# B&R Automation Studio project NAELD004C00R10L518F00 (part 49)

#### Act_InitLocal.st
```iecst
(** 2019-04-16 **)
ACTION Act_InitLocal:

	//Input Reference Link To Local Variable
	p_udiRstErr ACCESS ADR(udiRstErr);
	p_bEn ACCESS ADR(bEn);
	p_bDis ACCESS ADR(bDis);
	p_bRun ACCESS ADR(bRun);
	p_bStop ACCESS ADR(bStop);
	p_bStep ACCESS ADR(bStep);

	p_sProgNm ACCESS ADR(sProgNm);
	p_bNtSettingsLoadDone ACCESS ADR(bNtSettingsLoadDone);

	pa_bMagDis ACCESS ADR(a_bMagDis);
	p_bUnloadMag ACCESS ADR(bUnloadMag);
	p_bDSAllow ACCESS ADR(bDSAllow);
	p_bPullerRotCylPrep ACCESS ADR(bPullerRotCylPrep);
	p_bPullerNoRotCylExitStartLif ACCESS ADR(bPullerNoRotCylExitStartLif);
	p_diPullerExtMaxSlt ACCESS ADR(diPullerExtMaxSlt);
	p_diPullerExtMinSlt ACCESS ADR(diPullerExtMinSlt);
	p_bLifterSafeInitialize ACCESS ADR(bLifterSafeInitialize);

	p_bProdRcpCurrRcpTopToBtm ACCESS ADR(bProdRcpCurrRcpTopToBtm);
	p_diProdRcpCurrRcpPitch ACCESS ADR(diProdRcpCurrRcpPitch);

	p_bMagSetupDone1 ACCESS ADR(bMagSetupDone1);
	p_bMagSetupDone2 ACCESS ADR(bMagSetupDone2);
	p_bMagSetupDone3 ACCESS ADR(bMagSetupDone3);

	p_tyBufferStat1 ACCESS ADR(tyBufferStat1);
	p_tyBufferStat2 ACCESS ADR(tyBufferStat2);
	p_tyBufferStat3 ACCESS ADR(tyBufferStat3);

	p_bMagPresentSen1 ACCESS ADR(bMagPresentSen1);
	p_bMagPresentSen2 ACCESS ADR(bMagPresentSen2);
	p_bMagPresentSen3 ACCESS ADR(bMagPresentSen3);

	p_bBufferMagPresent1 ACCESS ADR(bBufferMagPresent1);
	p_bBufferMagPresent2 ACCESS ADR(bBufferMagPresent2);
	p_bBufferMagPresent3 ACCESS ADR(bBufferMagPresent3);

	p_dtBufferMagPresentTm1 ACCESS ADR(dtBufferMagPresentTm1);
	p_dtBufferMagPresentTm2 ACCESS ADR(dtBufferMagPresentTm2);
	p_dtBufferMagPresentTm3 ACCESS ADR(dtBufferMagPresentTm3);

	p_eLifterStat ACCESS ADR(eLifterStat);
	p_eLifterStatus ACCESS ADR(eLifterStatus);

	p_eBufferStat1 ACCESS ADR(eBufferStat1);
	p_eBufferStatus1 ACCESS ADR(eBufferStatus1);

	p_eBufferStat2 ACCESS ADR(eBufferStat2);
	p_eBufferStatus2 ACCESS ADR(eBufferStatus2);

	p_eBufferStat3 ACCESS ADR(eBufferStat3);
	p_eBufferStatus3 ACCESS ADR(eBufferStatus3);

	p_eDSSMEMAStat1 ACCESS ADR(eDSSMEMAStat1);
	p_eDSSMEMAStatus1 ACCESS ADR(eDSSMEMAStatus1);
	p_bDSSMEMAConvStart1 ACCESS ADR(bDSSMEMAConvStart1);

	p_eDSSMEMAStat2 ACCESS ADR(eDSSMEMAStat2);
	p_eDSSMEMAStatus2 ACCESS ADR(eDSSMEMAStatus2);
	p_bDSSMEMAConvStart2 ACCESS ADR(bDSSMEMAConvStart2);

	p_eDSSMEMAStat3 ACCESS ADR(eDSSMEMAStat3);
	p_eDSSMEMAStatus3 ACCESS ADR(eDSSMEMAStatus3);
	p_bDSSMEMAConvStart3 ACCESS ADR(bDSSMEMAConvStart3);

	p_diBufferNxtUnloadSlt1 ACCESS ADR(diBufferNxtUnloadSlt1);
	p_diBufferNxtUnloadSlt2 ACCESS ADR(diBufferNxtUnloadSlt2);
	p_diBufferNxtUnloadSlt3 ACCESS ADR(diBufferNxtUnloadSlt3);

END_ACTION
```

#### Act_Link.st
```iecst
(** 2018-12-11 **)
ACTION Act_Link:
	p_bLifterSafeInitialize := p_bLinkPullerRetRS AND p_bLinkInShutterCloRS;

END_ACTION
```

#### Init.st
```iecst
(** 2019-03-25 **)
PROGRAM _INIT

	(* Always Change If Project Change *)

	//Pass Address To Global Address For External Use
	//Action, State & Status

	//Alarm
	p_OpsLifMagLDAlmData	:= ADR(tyAlmData);
	p_OpsLifMagLDAlmData1	:= ADR(tyAlmData1);

	//Output
	p_OpsLifMagLDStepTxt	:= ADR(sStepTxt);
	p_OpsLifMagLDPaused		:= ADR(bPaused);

	p_OpsLifMagLDLifterAct		:= ADR(eLifterAct);
	p_OpsLifMagLDBufferAct1		:= ADR(eBufferAct1);
	p_OpsLifMagLDBufferAct2		:= ADR(eBufferAct2);
	p_OpsLifMagLDBufferAct3		:= ADR(eBufferAct3);
	p_OpsLifMagLDDSSMEMAAct1	:= ADR(eDSSMEMAAct1);
	p_OpsLifMagLDDSSMEMAAct2	:= ADR(eDSSMEMAAct2);
	p_OpsLifMagLDDSSMEMAAct3	:= ADR(eDSSMEMAAct3);

	p_OpsLifMagLDGoUnloadSlt1	:= ADR(diGoUnloadSlt1);
	p_OpsLifMagLDGoUnloadSlt2	:= ADR(diGoUnloadSlt2);
	p_OpsLifMagLDGoUnloadSlt3	:= ADR(diGoUnloadSlt3);
	p_OpsLifMagLDMagNxtUnload	:= ADR(eMagNxtUnload);
	p_OpsLifMagLDBffrExitBrd	:= ADR(bBffrExitBrd);
	p_OpsLifMagLDUnloadingMov	:= ADR(bUnloadingMov);
	p_OpsLifMagLDUnloading		:= ADR(bUnloading);

	(* Always Change If Project Change *)

END_PROGRAM
```

#### Act_OpsInitial.st - Do Not Change!!!
```iecst
(** 2019-01-16 **)
ACTION Act_OpsInitial:

	eOpsStep		:= LifMagLDStepNA;
	eGotoOpsStep	:= LifMagLDStepInitLif;

	eOpsStep1		:= LifMagLDStep1NA;
	eGotoOpsStep1	:= LifMagLDStep1InitLif;

	eMagNxtUnload	:= MagNxtUnloadInvalid;
	bBffrExitBrd	:= FALSE;
	bUnloadingMov	:= FALSE;
	bUnloading		:= FALSE;

END_ACTION
```

#### Act_OpsRun.st
```iecst
(** 2019-04-16 **)
ACTION Act_OpsRun:

//	IF p_bPullerRotCylPrep = TRUE THEN
//		Act_OpsSubRun;
//	ELSE
		Act_OpsSubRun1;
//	END_IF

END_ACTION
```

#### Act_OpsInfo.st
```iecst
ACTION Act_OpsInfo:

	//Reset
	udiStatus1	:= 0;

	//Magazine Not Present
	a_bMagAllwMagPresent[1]	:= p_bMagPresentSen1;
	a_bMagAllwMagPresent[2]	:= p_bMagPresentSen2;
	a_bMagAllwMagPresent[3]	:= p_bMagPresentSen3;

	FOR udi := 1 TO 3 DO
		IF pa_bMagDis[udi] = FALSE AND a_bMagAllwMagPresent[udi] = TRUE THEN
			EXIT;
		END_IF
	END_FOR

	IF udi = 4 THEN
		IF (eOpsStep > LifMagLDStepInitLif) OR (eOpsStep1 > LifMagLDStep1InitLif) THEN
			udiStatus1	:= 10000;
		END_IF
	END_IF

	//Magazine Is Empty
	a_tyMagAllwBffrStat[1]	:= p_tyBufferStat1;
	a_tyMagAllwBffrStat[2]	:= p_tyBufferStat2;
	a_tyMagAllwBffrStat[3]	:= p_tyBufferStat3;

	FOR udi := 1 TO 3 DO
		IF pa_bMagDis[udi] = FALSE AND a_bMagAllwMagPresent[udi] = TRUE AND a_tyMagAllwBffrStat[udi].bBffrMty = TRUE THEN
			udiStatus1	:= 10001 + (udi - 1);
			EXIT;
		END_IF
	END_FOR

END_ACTION
```

#### Act_OpsRst.st - Do Not Change!!!
```iecst
(** 2019-03-25 **)
ACTION Act_OpsRst:

	udiStatus1	:= 0;

	eLifterAct		:= LifterActIdle;
	eBufferAct1		:= BufferActIdle;
	eBufferAct2		:= BufferActIdle;
	eBufferAct3		:= BufferActIdle;
	eDSSMEMAAct1	:= SMEMAActIdle;
	eDSSMEMAAct2	:= SMEMAActIdle;
	eDSSMEMAAct3	:= SMEMAActIdle;

END_ACTION
```

#### Act_OpsSubRun.st
```iecst
ACTION Act_OpsSubRun:

	(*Loader's Lifter Magazine Layout*)
	(*
		Direction: -->> LEFT TO RIGHT -->>

	     +----------+
	     |          |
	     |          |
	     |          |DS3 (Lif=PosCSlt)
	     |          |[Mag 3]
	     |          |
	     |          |DS2 (Lif=PosBSlt)
	     |          |[Mag 2]
	     |          |
	     |          |DS1 (Lif=PosASlt)
	     |          |[Mag 1]
	     |  Loader  |
	     +----------+

		Note: Program Action Called For Lifter As Shown Above
		      Setup Lifter Program Parameters Accordingly
	*)

	IF eGotoOpsStep <> eOpsStep THEN

		CASE eGotoOpsStep OF

			ELSE
				eOpsStep	:= eGotoOpsStep;

		END_CASE

	END_IF

	IF eOpsStep = eGotoOpsStep THEN

		IF bPaused = FALSE THEN

			CASE eOpsStep OF

				LifMagLDStepInitLif:
					sStepTxt	:= 'Initializing Lifter';

					IF p_bLifterSafeInitialize THEN
						eLifterAct	:= LifterActFullHm;

						IF p_eLifterStatus = Done AND p_eLifterStat = LifterActFullHm THEN
							eLifterAct	:= LifterActIdle;

							eGotoOpsStep	:= LifMagLDStepMagCmp;

							bPaused	:= p_bStop OR p_bStep;
						END_IF
					ELSE
						IF p_eLifterStat <> LifterActIdle THEN
							eLifterAct	:= LifterActStop;

							IF p_eLifterStatus = Done AND p_eLifterStat = LifterActStop THEN
								eLifterAct	:= LifterActIdle;

								bPaused	:= p_bStop OR p_bStep;
							END_IF
						ELSE
							bPaused	:= p_bStop OR p_bStep;
						END_IF
					END_IF

				LifMagLDStepMagCmp:
					sStepTxt	:= 'Comparing Magazine';

					a_bMagAllwMagSetupDone[1]	:= p_bMagSetupDone1;
					a_bMagAllwMagSetupDone[2]	:= p_bMagSetupDone2;
					a_bMagAllwMagSetupDone[3]	:= p_bMagSetupDone3;

					a_tyMagAllwBffrStat[1]	:= p_tyBufferStat1;
					a_tyMagAllwBffrStat[2]	:= p_tyBufferStat2;
					a_tyMagAllwBffrStat[3]	:= p_tyBufferStat3;

					a_bMagAllwMagPresent[1]	:= p_bBufferMagPresent1;
					a_bMagAllwMagPresent[2]	:= p_bBufferMagPresent2;
					a_bMagAllwMagPresent[3]	:= p_bBufferMagPresent3;

					a_udiMagAllwMagPresentTm[1]	:= DT_TO_UDINT(p_dtBufferMagPresentTm1);
					a_udiMagAllwMagPresentTm[2]	:= DT_TO_UDINT(p_dtBufferMagPresentTm2);
					a_udiMagAllwMagPresentTm[3]	:= DT_TO_UDINT(p_dtBufferMagPresentTm3);

					//Sorting Priority
					memset(ADR(a_udiMagAllwPriority), 0, SIZEOF(a_udiMagAllwPriority));

					FOR udi := 1 TO 3 DO
						udiCount	:= 3;
						udiCmpTm	:= a_udiMagAllwMagPresentTm[udi];

						FOR udi1 := 1 TO 3 DO
							IF a_udiMagAllwMagPresentTm[udi1] > udiCmpTm THEN
								udiCount	:= udiCount - 1;
							END_IF
						END_FOR

						a_udiMagAllwPriority[udi]	:= udiCount;
					END_FOR

					FOR udi := 3 TO 1 BY -1 DO
						FOR udi1 := 3 TO 1 BY -1 DO
							IF (udi <> udi1) AND (a_udiMagAllwPriority[udi] = a_udiMagAllwPriority[udi1]) THEN
								a_udiMagAllwPriority[udi1]	:= a_udiMagAllwPriority[udi1] - 1;
							END_IF
						END_FOR
					END_FOR

					//Checking Buffer Status
					memset(ADR(a_udiMagAllwSum), 0, SIZEOF(a_udiMagAllwSum));

					FOR udi := 1 TO 3 DO
						//Priority
						a_udiMagAllwSum[udi]	:= a_udiMagAllwSum[udi] + a_udiMagAllwPriority[udi];
						//Enable
						IF pa_bMagDis[udi] = FALSE THEN
							a_udiMagAllwSum[udi]	:= a_udiMagAllwSum[udi] + 1000;
						END_IF
						//Magazine Setup Complete
						IF a_bMagAllwMagSetupDone[udi] = TRUE THEN
							a_udiMagAllwSum[udi]	:= a_udiMagAllwSum[udi] + 1000;
						END_IF
						//Magazine Present
						IF a_bMagAllwMagPresent[udi] = TRUE THEN
							a_udiMagAllwSum[udi]	:= a_udiMagAllwSum[udi] + 1000;
						END_IF
						//Magazine Full
						IF a_tyMagAllwBffrStat[udi].bBffrFull = TRUE THEN
							a_udiMagAllwSum[udi]	:= a_udiMagAllwSum[udi] + 2500;
						END_IF
						//Magazine Available
						IF a_tyMagAllwBffrStat[udi].bBffrFull = FALSE AND a_tyMagAllwBffrStat[udi].bBffrMty = FALSE THEN
							a_udiMagAllwSum[udi]	:= a_udiMagAllwSum[udi] + 3000;
						END_IF

					END_FOR

					udiMagAllwGo	:= 99;

					FOR udi := 1 TO 3 DO
						//Enable + Magazine Setup Done + Magazine Present + Magazine Available
						IF a_udiMagAllwSum[udi] >= 6000 THEN

							IF udiMagAllwGo <> 99 THEN
								//Priority
								IF a_udiMagAllwSum[udi] < a_udiMagAllwSum[udiMagAllwGo] THEN
									udiMagAllwGo	:= udi;
								END_IF
							ELSE
								udiMagAllwGo	:= udi;
							END_IF

						END_IF

					END_FOR

					IF udiMagAllwGo = 99 THEN

						FOR udi := 1 TO 3 DO
							//Enable + Magazine Setup Done + Magazine Present + Magazine Full
							IF a_udiMagAllwSum[udi] >= 5500 THEN

								IF udiMagAllwGo <> 99 THEN
									//Priority
									IF a_udiMagAllwSum[udi] < a_udiMagAllwSum[udiMagAllwGo] THEN
										udiMagAllwGo	:= udi;
									END_IF
								ELSE
									udiMagAllwGo	:= udi;
								END_IF

							END_IF

						END_FOR

					END_IF

					IF (p_bDSAllow = TRUE) AND (udiMagAllwGo <> 99) THEN

						eMagNxtUnload	:= udiMagAllwGo;
						eGotoOpsStep	:= LifMagLDStepNxtUnloadBffr;

						IF eMagNxtUnload = MagNxtUnloadMag1 THEN
							p_tyLocalBufferStat ACCESS ADR(p_tyBufferStat1);
							p_bLocalBufferMagPresent ACCESS ADR(p_bBufferMagPresent1);
							p_dtLocalBufferMagPresentTm ACCESS ADR(p_dtBufferMagPresentTm1);

							p_eLocalBufferAct ACCESS ADR(eBufferAct1);
							p_eLocalBufferStat ACCESS ADR(p_eBufferStat1);
							p_eLocalBufferStatus ACCESS ADR(p_eBufferStatus1);

							p_eLocalDSSMEMAAct ACCESS ADR(eDSSMEMAAct1);
							p_eLocalDSSMEMAStat ACCESS ADR(p_eDSSMEMAStat1);
							p_eLocalDSSMEMAStatus ACCESS ADR(p_eDSSMEMAStatus1);
							p_bLocalDSSMEMAConvStart ACCESS ADR(p_bDSSMEMAConvStart1);

						ELSIF eMagNxtUnload = MagNxtUnloadMag2 THEN
							p_tyLocalBufferStat ACCESS ADR(p_tyBufferStat2);
							p_bLocalBufferMagPresent ACCESS ADR(p_bBufferMagPresent2);
							p_dtLocalBufferMagPresentTm ACCESS ADR(p_dtBufferMagPresentTm2);

							p_eLocalBufferAct ACCESS ADR(eBufferAct2);
							p_eLocalBufferStat ACCESS ADR(p_eBufferStat2);
							p_eLocalBufferStatus ACCESS ADR(p_eBufferStatus2);

							p_eLocalDSSMEMAAct ACCESS ADR(eDSSMEMAAct2);
							p_eLocalDSSMEMAStat ACCESS ADR(p_eDSSMEMAStat2);
							p_eLocalDSSMEMAStatus ACCESS ADR(p_eDSSMEMAStatus2);
							p_bLocalDSSMEMAConvStart ACCESS ADR(p_bDSSMEMAConvStart2);

						ELSIF eMagNxtUnload = MagNxtUnloadMag3 THEN
							p_tyLocalBufferStat ACCESS ADR(p_tyBufferStat3);
							p_bLocalBufferMagPresent ACCESS ADR(p_bBufferMagPresent3);
							p_dtLocalBufferMagPresentTm ACCESS ADR(p_dtBufferMagPresentTm3);

							p_eLocalBufferAct ACCESS ADR(eBufferAct3);
							p_eLocalBufferStat ACCESS ADR(p_eBufferStat3);
							p_eLocalBufferStatus ACCESS ADR(p_eBufferStatus3);

							p_eLocalDSSMEMAAct ACCESS ADR(eDSSMEMAAct3);
							p_eLocalDSSMEMAStat ACCESS ADR(p_eDSSMEMAStat3);
							p_eLocalDSSMEMAStatus ACCESS ADR(p_eDSSMEMAStatus3);
							p_bLocalDSSMEMAConvStart ACCESS ADR(p_bDSSMEMAConvStart3);

						END_IF

						bPaused	:= p_bStop OR p_bStep;

					ELSE

						eMagNxtUnload	:= MagNxtUnloadInvalid;

						bPaused	:= p_bStop;

					END_IF

					//Unload Magazine
					IF p_bUnloadMag = TRUE THEN
						eMagNxtUnload	:= MagNxtUnloadInvalid;
						eGotoOpsStep	:= LifMagLDStepLifMovUnloadMag;
					END_IF

				LifMagLDStepNxtUnloadBffr:
					sStepTxt	:= 'Computing Next Unload Buffer';

					p_eLocalBufferAct	:= BufferActNxtUnload;

					IF p_eLocalBufferStatus = Done AND p_eLocalBufferStat = BufferActNxtUnload THEN
						p_eLocalBufferAct	:= BufferActIdle;
						eGotoOpsStep		:= LifMagLDStepLifMov;

						bPaused	:= p_bStop OR p_bStep;

						//Unload Magazine
						IF p_bUnloadMag = TRUE THEN
							eMagNxtUnload	:= MagNxtUnloadInvalid;
							eGotoOpsStep	:= LifMagLDStepLifMovUnloadMag;
						END_IF

					END_IF

				LifMagLDStepLifMov:
					sStepTxt	:= 'Moving Lifter To Next Unload Position';

					diGoUnloadSlt1	:= p_diBufferNxtUnloadSlt1;
					diGoUnloadSlt2	:= p_diBufferNxtUnloadSlt2;
					diGoUnloadSlt3	:= p_diBufferNxtUnloadSlt3;

					IF eMagNxtUnload = MagNxtUnloadMag1 THEN
						eLifterAct	:= LifterActGoASltPos;

					ELSIF eMagNxtUnload = MagNxtUnloadMag2 THEN
						eLifterAct	:= LifterActGoBSltPos;

					ELSIF eMagNxtUnload = MagNxtUnloadMag3 THEN
						eLifterAct	:= LifterActGoCSltPos;

					ELSIF eMagNxtUnload = MagNxtUnloadInvalid THEN
						eGotoOpsStep	:= LifMagLDStepMagCmp;

						bPaused	:= p_bStop OR p_bStep;

						//Unload Magazine
						IF p_bUnloadMag = TRUE THEN
							eMagNxtUnload	:= MagNxtUnloadInvalid;
							eGotoOpsStep	:= LifMagLDStepLifMovUnloadMag;
						END_IF

					END_IF

					IF (p_eLifterStatus = Done AND p_eLifterStat = LifterActGoASltPos)
						OR (p_eLifterStatus = Done AND p_eLifterStat = LifterActGoBSltPos)
						OR (p_eLifterStatus = Done AND p_eLifterStat = LifterActGoCSltPos) THEN

						eLifterAct	:= LifterActIdle;

						eGotoOpsStep	:= LifMagLDStepBffrDSComm;

						bPaused	:= p_bStop OR p_bStep;

						//Unload Magazine
						IF p_bUnloadMag = TRUE THEN
							eMagNxtUnload	:= MagNxtUnloadInvalid;
							eGotoOpsStep	:= LifMagLDStepLifMovUnloadMag;
						END_IF

					END_IF

				LifMagLDStepBffrDSComm:
					sStepTxt	:= 'Communicating Buffer Downstream';

					p_eLocalDSSMEMAAct	:= SMEMAActRun;

					IF p_bLocalDSSMEMAConvStart = TRUE THEN
						eGotoOpsStep	:= LifMagLDStepBffrExitBrd;

					ELSIF p_bDSAllow = FALSE THEN
						p_eLocalDSSMEMAAct	:= SMEMAActIdle;
						eMagNxtUnload		:= MagNxtUnloadInvalid;
						eGotoOpsStep		:= LifMagLDStepMagCmp;

						bPaused	:= p_bStop OR p_bStep;

					ELSE

						IF p_bLocalBufferMagPresent = FALSE THEN	//Checking Magazine Present
							eMagNxtUnload	:= MagNxtUnloadInvalid;
							eGotoOpsStep	:= LifMagLDStepMagCmp;

							bPaused	:= p_bStop OR p_bStep;
						ELSIF pa_bMagDis[udiMagAllwGo] = TRUE THEN	//Checking Magazine Enable
							eMagNxtUnload	:= MagNxtUnloadInvalid;
							eGotoOpsStep	:= LifMagLDStepMagCmp;

							bPaused	:= p_bStop OR p_bStep;
						ELSE
							bPaused	:= p_bStop;
						END_IF

						//Unload Magazine
						IF p_bUnloadMag = TRUE THEN
							eMagNxtUnload	:= MagNxtUnloadInvalid;
							eGotoOpsStep	:= LifMagLDStepLifMovUnloadMag;

							bPaused	:= p_bStop OR p_bStep;
						END_IF

						IF (bPaused = TRUE) OR (eGotoOpsStep = LifMagLDStepMagCmp) OR (p_bUnloadMag = TRUE) THEN
							p_eLocalDSSMEMAAct	:= SMEMAActIdle;
						END_IF

					END_IF

				LifMagLDStepBffrExitBrd:
					IF p_bLocalDSSMEMAConvStart THEN
						sStepTxt	:= 'Transferring Board Out From Magazine';

						//Do Nothing
					END_IF

					IF p_eLocalDSSMEMAStatus = Done AND p_eLocalDSSMEMAStat = SMEMAActRun THEN
						p_eLocalDSSMEMAAct	:= SMEMAActIdle;
						eGotoOpsStep		:= LifMagLDStepUnloadBffr;
					END_IF

				LifMagLDStepUnloadBffr:
					sStepTxt	:= 'Unloading Buffer';

					p_eLocalBufferAct	:= BufferActUnload;

					IF p_eLocalBufferStatus = Done AND p_eLocalBufferStat = BufferActUnload THEN
						p_eLocalBufferAct	:= BufferActIdle;
						eMagNxtUnload		:= MagNxtUnloadInvalid;
						eGotoOpsStep		:= LifMagLDStepMagCmp;

						bPaused	:= p_bStop OR p_bStep;
					END_IF

				LifMagLDStepLifMovUnloadMag:
					sStepTxt	:= 'Moving Lifter To Unload Position';

					eLifterAct	:= LifterActGoAPos;

					IF p_eLifterStatus = Done AND p_eLifterStat = LifterActGoAPos THEN
						eLifterAct	:= LifterActIdle;

						eGotoOpsStep	:= LifMagLDStepUnloadMag;

						bPaused	:= p_bStop OR p_bStep;
					END_IF

				LifMagLDStepUnloadMag:
					sStepTxt	:= 'Unloading Magazine';

					IF p_bUnloadMag = FALSE THEN
						eGotoOpsStep	:= LifMagLDStepMagCmp;

						bPaused	:= p_bStop OR p_bStep;
					ELSE
						bPaused	:= p_bStop;
					END_IF

			END_CASE

		END_IF

	END_IF

	Act_OpsInfo;

	//Step
	bBffrExitBrd	:= eOpsStep = LifMagLDStepBffrExitBrd;
	bUnloadingMov	:= eOpsStep = LifMagLDStepLifMovUnloadMag;
	bUnloading		:= eOpsStep = LifMagLDStepUnloadMag;

END_ACTION
```

#### Act_OpsSubRun1.st
```iecst
ACTION Act_OpsSubRun1:

	(*Loader's Lifter Magazine Layout*)
	(*
		Direction: -->> LEFT TO RIGHT -->>

	     +----------+
	     |          |
	     |          |
	     |          |DS3 (Lif=PosCSlt)
	     |          |[Mag 3]
	     |          |
	     |          |DS2 (Lif=PosBSlt)
	     |          |[Mag 2]
	     |          |
	     |          |DS1 (Lif=PosASlt)
	     |          |[Mag 1]
	     |  Loader  |
	     +----------+

		Note: Program Action Called For Lifter As Shown Above
		      Setup Lifter Program Parameters Accordingly
	*)

	IF eGotoOpsStep1 <> eOpsStep1 THEN

		CASE eGotoOpsStep1 OF

			ELSE
				eOpsStep1	:= eGotoOpsStep1;

		END_CASE

	END_IF

	IF eOpsStep1 = eGotoOpsStep1 THEN

		IF bPaused = FALSE THEN

			CASE eOpsStep1 OF

				LifMagLDStep1InitLif:
					sStepTxt	:= 'Initializing Lifter';

					IF p_bLifterSafeInitialize THEN
						eLifterAct	:= LifterActFullHm;

						IF p_eLifterStatus = Done AND p_eLifterStat = LifterActFullHm THEN
							eLifterAct	:= LifterActIdle;

							eGotoOpsStep1	:= LifMagLDStep1MagCmp;

							bPaused	:= p_bStop OR p_bStep;
						END_IF
					ELSE
						IF p_eLifterStat <> LifterActIdle THEN
							eLifterAct	:= LifterActStop;

							IF p_eLifterStatus = Done AND p_eLifterStat = LifterActStop THEN
								eLifterAct	:= LifterActIdle;

								bPaused	:= p_bStop OR p_bStep;
							END_IF
						ELSE
							bPaused	:= p_bStop OR p_bStep;
						END_IF
					END_IF

				LifMagLDStep1MagCmp:
					sStepTxt	:= 'Comparing Magazine';

					a_bMagAllwMagSetupDone[1]	:= p_bMagSetupDone1;
					a_bMagAllwMagSetupDone[2]	:= p_bMagSetupDone2;
					a_bMagAllwMagSetupDone[3]	:= p_bMagSetupDone3;

					a_tyMagAllwBffrStat[1]	:= p_tyBufferStat1;
					a_tyMagAllwBffrStat[2]	:= p_tyBufferStat2;
					a_tyMagAllwBffrStat[3]	:= p_tyBufferStat3;

					a_bMagAllwMagPresent[1]	:= p_bBufferMagPresent1;
					a_bMagAllwMagPresent[2]	:= p_bBufferMagPresent2;
					a_bMagAllwMagPresent[3]	:= p_bBufferMagPresent3;

					a_udiMagAllwMagPresentTm[1]	:= DT_TO_UDINT(p_dtBufferMagPresentTm1);
					a_udiMagAllwMagPresentTm[2]	:= DT_TO_UDINT(p_dtBufferMagPresentTm2);
					a_udiMagAllwMagPresentTm[3]	:= DT_TO_UDINT(p_dtBufferMagPresentTm3);

					//Sorting Priority
					memset(ADR(a_udiMagAllwPriority), 0, SIZEOF(a_udiMagAllwPriority));

					FOR udi := 1 TO 3 DO
						udiCount	:= 3;
						udiCmpTm	:= a_udiMagAllwMagPresentTm[udi];

						FOR udi1 := 1 TO 3 DO
							IF a_udiMagAllwMagPresentTm[udi1] > udiCmpTm THEN
								udiCount	:= udiCount - 1;
							END_IF
						END_FOR

						a_udiMagAllwPriority[udi]	:= udiCount;
					END_FOR

					FOR udi := 3 TO 1 BY -1 DO
						FOR udi1 := 3 TO 1 BY -1 DO
							IF (udi <> udi1) AND (a_udiMagAllwPriority[udi] = a_udiMagAllwPriority[udi1]) THEN
								a_udiMagAllwPriority[udi1]	:= a_udiMagAllwPriority[udi1] - 1;
							END_IF
						END_FOR
					END_FOR

					//Checking Buffer Status
					memset(ADR(a_udiMagAllwSum), 0, SIZEOF(a_udiMagAllwSum));

					FOR udi := 1 TO 3 DO
						//Priority
						a_udiMagAllwSum[udi]	:= a_udiMagAllwSum[udi] + a_udiMagAllwPriority[udi];
						//Enable
						IF pa_bMagDis[udi] = FALSE THEN
							a_udiMagAllwSum[udi]	:= a_udiMagAllwSum[udi] + 1000;
						END_IF
						//Magazine Setup Complete
						IF a_bMagAllwMagSetupDone[udi] = TRUE THEN
							a_udiMagAllwSum[udi]	:= a_udiMagAllwSum[udi] + 1000;
						END_IF
						//Magazine Present
						IF a_bMagAllwMagPresent[udi] = TRUE THEN
							a_udiMagAllwSum[udi]	:= a_udiMagAllwSum[udi] + 1000;
						END_IF
						//Magazine Full
						IF a_tyMagAllwBffrStat[udi].bBffrFull = TRUE THEN
							a_udiMagAllwSum[udi]	:= a_udiMagAllwSum[udi] + 2500;
						END_IF
						//Magazine Available
						IF a_tyMagAllwBffrStat[udi].bBffrFull = FALSE AND a_tyMagAllwBffrStat[udi].bBffrMty = FALSE THEN
							a_udiMagAllwSum[udi]	:= a_udiMagAllwSum[udi] + 3000;
						END_IF

					END_FOR

					udiMagAllwGo	:= 99;

					FOR udi := 1 TO 3 DO
						//Enable + Magazine Setup Done + Magazine Present + Magazine Available
						IF a_udiMagAllwSum[udi] >= 6000 THEN

							IF udiMagAllwGo <> 99 THEN
								//Priority
								IF a_udiMagAllwSum[udi] < a_udiMagAllwSum[udiMagAllwGo] THEN
									udiMagAllwGo	:= udi;
								END_IF
							ELSE
								udiMagAllwGo	:= udi;
							END_IF

						END_IF

					END_FOR

					IF udiMagAllwGo = 99 THEN

						FOR udi := 1 TO 3 DO
							//Enable + Magazine Setup Done + Magazine Present + Magazine Full
							IF a_udiMagAllwSum[udi] >= 5500 THEN

								IF udiMagAllwGo <> 99 THEN
									//Priority
									IF a_udiMagAllwSum[udi] < a_udiMagAllwSum[udiMagAllwGo] THEN
										udiMagAllwGo	:= udi;
									END_IF
								ELSE
									udiMagAllwGo	:= udi;
								END_IF

							END_IF

						END_FOR

					END_IF

					IF (p_bDSAllow = TRUE) AND (udiMagAllwGo <> 99) THEN

						eMagNxtUnload	:= udiMagAllwGo;
						eGotoOpsStep1	:= LifMagLDStep1NxtUnloadBffr;

						IF eMagNxtUnload = MagNxtUnloadMag1 THEN
							p_tyLocalBufferStat ACCESS ADR(p_tyBufferStat1);
							p_bLocalBufferMagPresent ACCESS ADR(p_bBufferMagPresent1);
							p_dtLocalBufferMagPresentTm ACCESS ADR(p_dtBufferMagPresentTm1);

							p_eLocalBufferAct ACCESS ADR(eBufferAct1);
							p_eLocalBufferStat ACCESS ADR(p_eBufferStat1);
							p_eLocalBufferStatus ACCESS ADR(p_eBufferStatus1);

							p_eLocalDSSMEMAAct ACCESS ADR(eDSSMEMAAct1);
							p_eLocalDSSMEMAStat ACCESS ADR(p_eDSSMEMAStat1);
							p_eLocalDSSMEMAStatus ACCESS ADR(p_eDSSMEMAStatus1);
							p_bLocalDSSMEMAConvStart ACCESS ADR(p_bDSSMEMAConvStart1);

						ELSIF eMagNxtUnload = MagNxtUnloadMag2 THEN
							p_tyLocalBufferStat ACCESS ADR(p_tyBufferStat2);
							p_bLocalBufferMagPresent ACCESS ADR(p_bBufferMagPresent2);
							p_dtLocalBufferMagPresentTm ACCESS ADR(p_dtBufferMagPresentTm2);

							p_eLocalBufferAct ACCESS ADR(eBufferAct2);
							p_eLocalBufferStat ACCESS ADR(p_eBufferStat2);
							p_eLocalBufferStatus ACCESS ADR(p_eBufferStatus2);

							p_eLocalDSSMEMAAct ACCESS ADR(eDSSMEMAAct2);
							p_eLocalDSSMEMAStat ACCESS ADR(p_eDSSMEMAStat2);
							p_eLocalDSSMEMAStatus ACCESS ADR(p_eDSSMEMAStatus2);
							p_bLocalDSSMEMAConvStart ACCESS ADR(p_bDSSMEMAConvStart2);

						ELSIF eMagNxtUnload = MagNxtUnloadMag3 THEN
							p_tyLocalBufferStat ACCESS ADR(p_tyBufferStat3);
							p_bLocalBufferMagPresent ACCESS ADR(p_bBufferMagPresent3);
							p_dtLocalBufferMagPresentTm ACCESS ADR(p_dtBufferMagPresentTm3);

							p_eLocalBufferAct ACCESS ADR(eBufferAct3);
							p_eLocalBufferStat ACCESS ADR(p_eBufferStat3);
							p_eLocalBufferStatus ACCESS ADR(p_eBufferStatus3);

							p_eLocalDSSMEMAAct ACCESS ADR(eDSSMEMAAct3);
							p_eLocalDSSMEMAStat ACCESS ADR(p_eDSSMEMAStat3);
							p_eLocalDSSMEMAStatus ACCESS ADR(p_eDSSMEMAStatus3);
							p_bLocalDSSMEMAConvStart ACCESS ADR(p_bDSSMEMAConvStart3);

						END_IF

						bPaused	:= p_bStop OR p_bStep;

					ELSE

						eMagNxtUnload	:= MagNxtUnloadInvalid;

						bPaused	:= p_bStop;

					END_IF

					//Unload Magazine
					IF p_bUnloadMag = TRUE THEN
						eMagNxtUnload	:= MagNxtUnloadInvalid;
						eGotoOpsStep1	:= LifMagLDStep1LifMovUnloadMag;
					END_IF

				LifMagLDStep1NxtUnloadBffr:
					sStepTxt	:= 'Computing Next Unload Buffer';

					p_eLocalBufferAct	:= BufferActNxtUnload;

					IF p_eLocalBufferStatus = Done AND p_eLocalBufferStat = BufferActNxtUnload THEN
						p_eLocalBufferAct	:= BufferActIdle;
						IF p_bPullerRotCylPrep = FALSE THEN
							eGotoOpsStep1		:= LifMagLDStep1PreLifMov;
						ELSE
							IF p_bLinkInShutterExtended THEN
								eGotoOpsStep1		:= LifMagLDStep1LifMov;
							END_IF
						END_IF
						bPaused	:= p_bStop OR p_bStep;

						//Unload Magazine
						IF p_bUnloadMag = TRUE THEN
							eMagNxtUnload	:= MagNxtUnloadInvalid;
							eGotoOpsStep1	:= LifMagLDStep1LifMovUnloadMag;
						END_IF

					END_IF

				LifMagLDStep1LifMov:
					sStepTxt	:= 'Moving Lifter To Next Unload Position';

					diGoUnloadSlt1	:= p_diBufferNxtUnloadSlt1;
					diGoUnloadSlt2	:= p_diBufferNxtUnloadSlt2;
					diGoUnloadSlt3	:= p_diBufferNxtUnloadSlt3;

					IF eMagNxtUnload = MagNxtUnloadMag1 THEN
						eLifterAct	:= LifterActGoASltPos;

					ELSIF eMagNxtUnload = MagNxtUnloadMag2 THEN
						eLifterAct	:= LifterActGoBSltPos;

					ELSIF eMagNxtUnload = MagNxtUnloadMag3 THEN
						eLifterAct	:= LifterActGoCSltPos;

					ELSIF eMagNxtUnload = MagNxtUnloadInvalid THEN
						eGotoOpsStep1	:= LifMagLDStep1MagCmp;

						bPaused	:= p_bStop OR p_bStep;

						//Unload Magazine
						IF p_bUnloadMag = TRUE THEN
							eMagNxtUnload	:= MagNxtUnloadInvalid;
							eGotoOpsStep1	:= LifMagLDStep1LifMovUnloadMag;
						END_IF

					END_IF

					IF (p_eLifterStatus = Done AND p_eLifterStat = LifterActGoASltPos)
						OR (p_eLifterStatus = Done AND p_eLifterStat = LifterActGoBSltPos)
						OR (p_eLifterStatus = Done AND p_eLifterStat = LifterActGoCSltPos) THEN

						eLifterAct	:= LifterActIdle;

						eGotoOpsStep1	:= LifMagLDStep1BffrDSComm;

						bPaused	:= p_bStop OR p_bStep;

						//Unload Magazine
						IF p_bUnloadMag = TRUE THEN
							eMagNxtUnload	:= MagNxtUnloadInvalid;
							eGotoOpsStep1	:= LifMagLDStep1LifMovUnloadMag;
						END_IF

					END_IF

				LifMagLDStep1PreLifMov:
					sStepTxt	:= 'Pre-Moving Lifter To Next Unload Position';

					IF p_bProdRcpCurrRcpTopToBtm THEN

						IF p_diBufferNxtUnloadSlt1 >= p_diPullerExtMaxSlt THEN
							eStatus		:= Error;
							udiStatus	:= 10004;	//Lifter Pre-Exit Position Are Invalid
						ELSE
							IF (p_diBufferNxtUnloadSlt1 + p_diProdRcpCurrRcpPitch) > p_diPullerExtMaxSlt THEN
								diGoUnloadSlt1	:= p_diPullerExtMaxSlt;
							ELSE
								//	diGoUnloadSlt1	:= p_diBufferNxtUnloadSlt1 + p_diProdRcpCurrRcpPitch;
								IF p_diProdRcpCurrRcpPitch <= 4 THEN
									diGoUnloadSlt1	:= p_diBufferNxtUnloadSlt1 + p_diProdRcpCurrRcpPitch;
								ELSE
									diGoUnloadSlt1	:= p_diBufferNxtUnloadSlt1 + 4;
								END_IF
							END_IF
						END_IF

						IF p_diBufferNxtUnloadSlt2 >= p_diPullerExtMaxSlt THEN
							eStatus		:= Error;
							udiStatus	:= 10004;	//Lifter Pre-Exit Position Are Invalid
						ELSE
							IF (p_diBufferNxtUnloadSlt2 + p_diProdRcpCurrRcpPitch) > p_diPullerExtMaxSlt THEN
								diGoUnloadSlt2	:= p_diPullerExtMaxSlt;
							ELSE
								//	diGoUnloadSlt2	:= p_diBufferNxtUnloadSlt2 + p_diProdRcpCurrRcpPitch;
								IF p_diProdRcpCurrRcpPitch <= 4 THEN
									diGoUnloadSlt2	:= p_diBufferNxtUnloadSlt2 + p_diProdRcpCurrRcpPitch;
								ELSE
									diGoUnloadSlt2	:= p_diBufferNxtUnloadSlt2 + 4;
								END_IF
							END_IF
						END_IF

						IF p_diBufferNxtUnloadSlt3 >= p_diPullerExtMaxSlt THEN
							eStatus		:= Error;
							udiStatus	:= 10004;	//Lifter Pre-Exit Position Are Invalid
						ELSE
							IF (p_diBufferNxtUnloadSlt3 + p_diProdRcpCurrRcpPitch) > p_diPullerExtMaxSlt THEN
								diGoUnloadSlt3	:= p_diPullerExtMaxSlt;
							ELSE
								//	diGoUnloadSlt3	:= p_diBufferNxtUnloadSlt3 + p_diProdRcpCurrRcpPitch;
								IF p_diProdRcpCurrRcpPitch <= 4 THEN
									diGoUnloadSlt3	:= p_diBufferNxtUnloadSlt3 + p_diProdRcpCurrRcpPitch;
								ELSE
									diGoUnloadSlt3	:= p_diBufferNxtUnloadSlt3 + 4;
								END_IF
							END_IF
						END_IF

					ELSE

						IF p_diBufferNxtUnloadSlt1 <= p_diPullerExtMinSlt THEN
							eStatus		:= Error;
							udiStatus	:= 10004;	//Lifter Pre-Exit Position Are Invalid
						ELSE
							IF (p_diBufferNxtUnloadSlt1 - p_diProdRcpCurrRcpPitch) < p_diPullerExtMinSlt THEN
								diGoUnloadSlt1	:= p_diPullerExtMinSlt;
							ELSE
								diGoUnloadSlt1	:= p_diBufferNxtUnloadSlt1 - p_diProdRcpCurrRcpPitch;
							END_IF
						END_IF

						IF p_diBufferNxtUnloadSlt2 <= p_diPullerExtMinSlt THEN
							eStatus		:= Error;
							udiStatus	:= 10004;	//Lifter Pre-Exit Position Are Invalid
						ELSE
							IF (p_diBufferNxtUnloadSlt2 - p_diProdRcpCurrRcpPitch) < p_diPullerExtMinSlt THEN
								diGoUnloadSlt2	:= p_diPullerExtMinSlt;
							ELSE
								diGoUnloadSlt2	:= p_diBufferNxtUnloadSlt2 - p_diProdRcpCurrRcpPitch;
							END_IF
						END_IF

						IF p_diBufferNxtUnloadSlt3 <= p_diPullerExtMinSlt THEN
							eStatus		:= Error;
							udiStatus	:= 10004;	//Lifter Pre-Exit Position Are Invalid
						ELSE
							IF (p_diBufferNxtUnloadSlt3 - p_diProdRcpCurrRcpPitch) < p_diPullerExtMinSlt THEN
								diGoUnloadSlt3	:= p_diPullerExtMinSlt;
							ELSE
								diGoUnloadSlt3	:= p_diBufferNxtUnloadSlt3 - p_diProdRcpCurrRcpPitch;
							END_IF
						END_IF

					END_IF

					IF eMagNxtUnload = MagNxtUnloadMag1 THEN
						eLifterAct	:= LifterActGoASltPos;

					ELSIF eMagNxtUnload = MagNxtUnloadMag2 THEN
						eLifterAct	:= LifterActGoBSltPos;

					ELSIF eMagNxtUnload = MagNxtUnloadMag3 THEN
						eLifterAct	:= LifterActGoCSltPos;

					ELSIF eMagNxtUnload = MagNxtUnloadInvalid THEN
						eGotoOpsStep1	:= LifMagLDStep1MagCmp;

						bPaused	:= p_bStop OR p_bStep;

						//Unload Magazine
						IF p_bUnloadMag = TRUE THEN
							eMagNxtUnload	:= MagNxtUnloadInvalid;
							eGotoOpsStep1	:= LifMagLDStep1LifMovUnloadMag;
						END_IF

					END_IF

					IF (p_eLifterStatus = Done AND p_eLifterStat = LifterActGoASltPos)
						OR (p_eLifterStatus = Done AND p_eLifterStat = LifterActGoBSltPos)
						OR (p_eLifterStatus = Done AND p_eLifterStat = LifterActGoCSltPos) THEN

						eLifterAct	:= LifterActIdle;

						eGotoOpsStep1	:= LifMagLDStep1BffrDSComm;

						bPaused	:= p_bStop OR p_bStep;

						//Unload Magazine
						IF p_bUnloadMag = TRUE THEN
							eMagNxtUnload	:= MagNxtUnloadInvalid;
							eGotoOpsStep1	:= LifMagLDStep1LifMovUnloadMag;
						END_IF

					END_IF

				LifMagLDStep1BffrDSComm:
					sStepTxt	:= 'Communicating Buffer Downstream';

					p_eLocalDSSMEMAAct	:= SMEMAActRun;

					IF p_bLocalDSSMEMAConvStart = TRUE THEN
						IF p_bPullerRotCylPrep = FALSE THEN
							eGotoOpsStep1	:= LifMagLDStep1BffrExitLifMovWait;
						ELSE
							eGotoOpsStep1	:= LifMagLDStep1BffrExitBrd;
						END_IF

					ELSIF p_bDSAllow = FALSE THEN
						p_eLocalDSSMEMAAct	:= SMEMAActIdle;
						eMagNxtUnload		:= MagNxtUnloadInvalid;
						eGotoOpsStep1		:= LifMagLDStep1MagCmp;

						bPaused	:= p_bStop OR p_bStep;

					ELSE

						IF p_bLocalBufferMagPresent = FALSE THEN	//Checking Magazine Present
							eMagNxtUnload	:= MagNxtUnloadInvalid;
							eGotoOpsStep1	:= LifMagLDStep1MagCmp;

							bPaused	:= p_bStop OR p_bStep;
						ELSIF pa_bMagDis[udiMagAllwGo] = TRUE THEN	//Checking Magazine Enable
							eMagNxtUnload	:= MagNxtUnloadInvalid;
							eGotoOpsStep1	:= LifMagLDStep1MagCmp;

							bPaused	:= p_bStop OR p_bStep;
						ELSE
							bPaused	:= p_bStop;
						END_IF

						//Unload Magazine
						IF p_bUnloadMag = TRUE THEN
							eMagNxtUnload	:= MagNxtUnloadInvalid;
							eGotoOpsStep1	:= LifMagLDStep1LifMovUnloadMag;

							bPaused	:= p_bStop OR p_bStep;
						END_IF

						IF (bPaused = TRUE) OR (eGotoOpsStep1 = LifMagLDStep1MagCmp) OR (p_bUnloadMag = TRUE) THEN
							p_eLocalDSSMEMAAct	:= SMEMAActIdle;
						END_IF

					END_IF

				LifMagLDStep1BffrExitLifMovWait:
					sStepTxt	:= 'Waiting For Lifter Start Move Signal';

					IF p_bPullerNoRotCylExitStartLif THEN
						eGotoOpsStep1	:= LifMagLDStep1BffrExitLifMov;
					END_IF

				LifMagLDStep1BffrExitLifMov:
					sStepTxt	:= 'Moving Lifter To Next Unload Position';

					diGoUnloadSlt1	:= p_diBufferNxtUnloadSlt1;
					diGoUnloadSlt2	:= p_diBufferNxtUnloadSlt2;
					diGoUnloadSlt3	:= p_diBufferNxtUnloadSlt3;

					IF eMagNxtUnload = MagNxtUnloadMag1 THEN
						eLifterAct	:= LifterActGoASltPos;

					ELSIF eMagNxtUnload = MagNxtUnloadMag2 THEN
						eLifterAct	:= LifterActGoBSltPos;

					ELSIF eMagNxtUnload = MagNxtUnloadMag3 THEN
						eLifterAct	:= LifterActGoCSltPos;

					ELSIF eMagNxtUnload = MagNxtUnloadInvalid THEN
						eStatus		:= Error;
						udiStatus	:= 10005;	//Lifter Exit Position Are Invalid

					END_IF

					IF (p_eLifterStatus = Done AND p_eLifterStat = LifterActGoASltPos)
						OR (p_eLifterStatus = Done AND p_eLifterStat = LifterActGoBSltPos)
						OR (p_eLifterStatus = Done AND p_eLifterStat = LifterActGoCSltPos) THEN

						eLifterAct	:= LifterActIdle;

						eGotoOpsStep1	:= LifMagLDStep1BffrExitBrd;

					END_IF

				LifMagLDStep1BffrExitBrd:
					IF p_bLocalDSSMEMAConvStart THEN
						sStepTxt	:= 'Transferring Board Out From Magazine';

						//Do Nothing
					END_IF

					IF p_eLocalDSSMEMAStatus = Done AND p_eLocalDSSMEMAStat = SMEMAActRun THEN
						p_eLocalDSSMEMAAct	:= SMEMAActIdle;
						eGotoOpsStep1		:= LifMagLDStep1UnloadBffr;
					END_IF

				LifMagLDStep1UnloadBffr:
					sStepTxt	:= 'Unloading Buffer';

					p_eLocalBufferAct	:= BufferActUnload;

					IF p_eLocalBufferStatus = Done AND p_eLocalBufferStat = BufferActUnload THEN
						p_eLocalBufferAct	:= BufferActIdle;
						eMagNxtUnload		:= MagNxtUnloadInvalid;
						eGotoOpsStep1		:= LifMagLDStep1MagCmp;

						bPaused	:= p_bStop OR p_bStep;
					END_IF

				LifMagLDStep1LifMovUnloadMag:
					sStepTxt	:= 'Moving Lifter To Unload Position';

					eLifterAct	:= LifterActGoAPos;

					IF p_eLifterStatus = Done AND p_eLifterStat = LifterActGoAPos THEN
						eLifterAct	:= LifterActIdle;

						eGotoOpsStep1	:= LifMagLDStep1UnloadMag;

						bPaused	:= p_bStop OR p_bStep;
					END_IF

				LifMagLDStep1UnloadMag:
					sStepTxt	:= 'Unloading Magazine';

					IF p_bUnloadMag = FALSE THEN
						eGotoOpsStep1	:= LifMagLDStep1MagCmp;

						bPaused	:= p_bStop OR p_bStep;
					ELSE
						bPaused	:= p_bStop;
					END_IF

			END_CASE

		END_IF

	END_IF

	Act_OpsInfo;

	//Step
	bBffrExitBrd	:= eOpsStep1 = LifMagLDStep1BffrExitBrd;
	bUnloadingMov	:= eOpsStep1 = LifMagLDStep1LifMovUnloadMag;
	bUnloading		:= eOpsStep1 = LifMagLDStep1UnloadMag;

END_ACTION
```

### AGV.typ - Do Not Change!!!
```iecst
(*2018-12-13*)
(**)
(*Action*)

TYPE
	eAGVMagAction :
		(
		AGVMagActIdle,
		AGVMagActEnter,
		AGVMagActExit
		);
	tyTagDTMagToAGV : 	STRUCT
		bEStopErr : BOOL;
		bCI1MagazineEmpty : BOOL;
		bCI1Rdy : BOOL;
		bCI1Auto : BOOL;
		bCI1Occupied : BOOL;
		bCI1Running : BOOL;
		bCI1IncorrectMagazineModel : BOOL;
		bCI2MagazineEmpty : BOOL;
		bCI2Rdy : BOOL;
		bCI2Auto : BOOL;
		bCI2Occupied : BOOL;
		bCI2Running : BOOL;
		bCI2IncorrectMagazineModel : BOOL;
		bCI3MagazineEmpty : BOOL;
		bCI3Rdy : BOOL;
		bCI3Auto : BOOL;
		bCI3Occupied : BOOL;
		bCI3Running : BOOL;
		bCI3IncorrectMagazineModel : BOOL;
		bCI4MagazineEmpty : BOOL;
		bCI4Rdy : BOOL;
		bCI4Auto : BOOL;
		bCI4Occupied : BOOL;
		bCI4Running : BOOL;
		bCI4IncorrectMagazineModel : BOOL;
	END_STRUCT;
	tyTagAGVToDTMag : 	STRUCT
		bVEHInPos1 : BOOL;
		bVEHInPos2 : BOOL;
		bVEHInPos3 : BOOL;
		bVEHInPos4 : BOOL;
		bVEHAuto : BOOL;
		bVEH1Occupied : BOOL;
		bVEH2Occupied : BOOL;
		bVEH3Occupied : BOOL;
		bVEH4Occupied : BOOL;
		bVEHRunning : BOOL;
	END_STRUCT;
	tyStatToMES : 	STRUCT
		sMachineName : STRING[30];
		bActive : BOOL;
		bAuto_Run : BOOL;
		bError : BOOL;
		bWarning : BOOL;
		nNumberOfPlatforms : USINT;
		tyTagStatOfPlatforms : ARRAY[1..4]OF tyStatPlatform;
	END_STRUCT;
	tyStatFromMES : 	STRUCT
		sMESName : STRING[30];
		bActive : BOOL;
		tyTagStatOfPlatforms : ARRAY[1..4]OF tyStatPlatformFromMES;
	END_STRUCT;
	tyStatPlatform : 	STRUCT
		bMagLoaded : BOOL;
		bReqAIVToBring : BOOL;
		bReqAIVToGet : BOOL;
		bReadRFID : BOOL;
		bWriteRFID : BOOL;
		bError : BOOL;
		bSizeLarge : BOOL;
		bReady : BOOL;
		bAvailable : BOOL;
	END_STRUCT;
	tyStatPlatformFromMES : 	STRUCT
		iAcceptCondition : INT;
		bRFIDWriteComplete : BOOL;
		bError : BOOL;
		bSizeLarge : BOOL;
		bReady : BOOL;
		bAvailable : BOOL;
	END_STRUCT;
END_TYPE
```

### Program Logical/AGVCom/AGV (IEC, version 1.00.0) - 1.00.0 - NtSMEMA v5.00.0

#### Init.st - Change By Project
```iecst
(** 2019-01-20 **)
PROGRAM _INIT

	(* Always Change If Project Change *)

	sProgNm	:= 'AGV';

	//Physical Configuration

	//Pass Address To Global Address For External Use
	//Action, State & Status
	p_AGVStat		     := ADR(eStat);
	p_AGVStatus		     := ADR(eStatus);
	p_AGVStatTxt	     := ADR(sStatTxt);

	//Alarm
	p_AGVAlmData		 := ADR(tyAlmData);
	p_AGVAlmData1		 := ADR(tyAlmData1);
	//Output
	p_AGVTagAGVToDTMag 	 := ADR(tyAGVToDTMag);
	p_AGVOnline			 := ADR(bInternalAGVOnline);
	p_MachineOnline		 := ADR(bMachineOnline);
	p_DTMagToAGV 		 := ADR(tyDTMagToAGV);
	p_AGVSimulationOn 	 := ADR(bInternalAGVSimulateOn);
	p_TagToMes			 := ADR(tyTagToMes);
	p_TagFromMes		 := ADR(tyTagFromMes);
	p_FleetManagerActive := ADR(bFleetManagerActive);

	//For Siemen
	p_TagToMesMagConv1		:= ADR(tyTagToMes.tyTagStatOfPlatforms[1]);
	p_TagToMesMagConv2		:= ADR(tyTagToMes.tyTagStatOfPlatforms[2]);
	p_TagToMesMagConv3		:= ADR(tyTagToMes.tyTagStatOfPlatforms[3]);
	p_TagFromMesMagConv1	:= ADR(tyTagFromMes.tyTagStatOfPlatforms[1]);
	p_TagFromMesMagConv2	:= ADR(tyTagFromMes.tyTagStatOfPlatforms[2]);
	p_TagFromMesMagConv3	:= ADR(tyTagFromMes.tyTagStatOfPlatforms[3]);

	(* Always Change If Project Change *)

END_PROGRAM
```

#### Act_InitGlobal.st - Change By Project
```iecst
(** 2018-12-08 **)
ACTION Act_InitGlobal:

	(* Always Change If Project Change *)

	//Pass Data To Link
	p_bLinkSafetyRlySig ACCESS p_DISafetyRlySig;
	p_bLinkCoverSWSig ACCESS p_DICoverSWSig;
	p_bLinkAlarmWarning ACCESS p_AlarmWarning;
	p_bLinkAlarmInfo ACCESS p_AlarmInfo;
	p_bLinkError ACCESS p_AlarmErr;
	p_eLinkLDMag ACCESS p_NtParamProjMag;
	p_eLinkAGVComProtocol ACCESS p_McParamAGVComProtocol;

	//Pass Data To Internal Use
	p_bOpsRun ACCESS p_OpsRun;
	p_bManual ACCESS p_UIUIMnlMod;

	p_bPrep ACCESS p_NtParamProjAGVPrep;
	p_bEn ACCESS p_McParamAGVComEn;
	p_tyDTMagToAGV1 ACCESS p_AGVMag1DTMagToAGV;
	p_tyDTMagToAGV2 ACCESS p_AGVMag2DTMagToAGV;
	p_tyDTMagToAGV3 ACCESS p_AGVMag3DTMagToAGV;
	p_tyDTMagToAGV4 ACCESS p_AGVMag4DTMagToAGV;
	p_udiRstErr	ACCESS p_RstErrReset;
	p_bNtSettingsLoadDone ACCESS p_StartupNtSettingsLoadDone;
	p_bIncorrectMagazine1 ACCESS p_OpsMagConvLD1IncorrectMagModel;
	p_bIncorrectMagazine2 ACCESS p_OpsMagConvLD2IncorrectMagModel;
	p_bIncorrectMagazine3 ACCESS p_OpsMagConvLD3IncorrectMagModel;
	p_bIncorrectMagazine4 ACCESS p_OpsMagConvLD4IncorrectMagModel;

	p_tyUIAGVToDTMagSimulateData ACCESS p_UIAGVSimulateSig;
	p_bUIAGVOnline ACCESS p_UIAGVSimulateOnline;
	p_bUIAGVSimulationOn ACCESS p_UIAGVSimulationOn;

	p_sJobNo ACCESS p_NtParamJobNo;

	p_bAGVRdyEnter1 ACCESS p_AGVMag1RdyEnter;
	p_bAGVRdyExit1 ACCESS p_AGVMag1RdyExit;
	p_bAGVRdyEnter2 ACCESS p_AGVMag2RdyEnter;
	p_bAGVRdyExit2 ACCESS p_AGVMag2RdyExit;
	p_bAGVRdyEnter3 ACCESS p_AGVMag3RdyEnter;
	p_bAGVRdyExit3 ACCESS p_AGVMag3RdyExit;
	p_bAGVRdyEnter4 ACCESS p_AGVMag4RdyEnter;
	p_bAGVRdyExit4 ACCESS p_AGVMag4RdyExit;

	p_bRequestToBring1 ACCESS p_Buffer1MagRemoved;
	p_bRequestToBring2 ACCESS p_Buffer2MagRemoved;
	p_bRequestToBring3 ACCESS p_Buffer3MagRemoved;
	p_bRequestToBring4 ACCESS p_Buffer4MagRemoved;
	p_bRequestToGet1 ACCESS p_DSSOT1DBA;
	p_bRequestToGet2 ACCESS p_DSSOT2DBA;
	p_bRequestToGet3 ACCESS p_DSSOT3DBA;
	p_bRequestToGet4 ACCESS p_DSSOT4DBA;

	p_bDIFleetManagerActive ACCESS p_DIFleetManagerActive;

	p_bUISOTMagError1	ACCESS p_UISOTMagErr1;
	p_bUISOTMagError2	ACCESS p_UISOTMagErr2;
	p_bUISOTMagError3	ACCESS p_UISOTMagErr3;
	p_bUISOTMagError4	ACCESS p_UISOTMagErr4;

	p_bUISOTMagReady1	ACCESS p_UISOTMagRdy1;
	p_bUISOTMagReady2	ACCESS p_UISOTMagRdy2;
	p_bUISOTMagReady3	ACCESS p_UISOTMagRdy3;
	p_bUISOTMagReady4	ACCESS p_UISOTMagRdy4;

	p_bUISOTMagAvailable1	ACCESS p_UISOTMagAvail1;
	p_bUISOTMagAvailable2	ACCESS p_UISOTMagAvail2;
	p_bUISOTMagAvailable3	ACCESS p_UISOTMagAvail3;
	p_bUISOTMagAvailable4	ACCESS p_UISOTMagAvail4;

	p_bUISOTMagSizeLarge1	ACCESS p_UISOTMagSLarge1;
	p_bUISOTMagSizeLarge2	ACCESS p_UISOTMagSLarge2;
	p_bUISOTMagSizeLarge3 ACCESS p_UISOTMagSLarge3;
	p_bUISOTMagSizeLarge4	ACCESS p_UISOTMagSLarge4;

	p_bUIRequestToBring1 ACCESS p_UIAIVReqBring1;
	p_bUIRequestToBring2 ACCESS p_UIAIVReqBring2;
	p_bUIRequestToBring3 ACCESS p_UIAIVReqBring3;
	p_bUIRequestToBring4 ACCESS p_UIAIVReqBring4;

	p_bUIRequestToGet1 ACCESS p_UIAIVReqGet1;
	p_bUIRequestToGet2 ACCESS p_UIAIVReqGet2;
	p_bUIRequestToGet3 ACCESS p_UIAIVReqGet3;
	p_bUIRequestToGet4 ACCESS p_UIAIVReqGet4;

	p_eAGVComProtocol ACCESS p_McParamAGVComProtocol;

	p_bSOTMagReady1 ACCESS p_USSOT1USB;
	p_bSOTMagReady2 ACCESS p_USSOT2USB;
	p_bSOTMagReady3 ACCESS p_USSOT3USB;
	p_bSOTMagReady4 ACCESS p_USSOT4USB;

	p_bSOTMagError1 ACCESS p_AlarmErr;
	p_bSOTMagError2 ACCESS p_AlarmErr;
	p_bSOTMagError3 ACCESS p_AlarmErr;
	p_bSOTMagError4 ACCESS p_AlarmErr;

	p_bSOTMagAvailable1 ACCESS p_DSSOT1DBA;
	p_bSOTMagAvailable2 ACCESS p_DSSOT2DBA;
	p_bSOTMagAvailable3 ACCESS p_DSSOT3DBA;
	p_bSOTMagAvailable4 ACCESS p_DSSOT4DBA;

	p_bSOTMagSizeLarge1 ACCESS p_DSSOT1MagSizeLarge;
	p_bSOTMagSizeLarge2 ACCESS p_DSSOT2MagSizeLarge;
	p_bSOTMagSizeLarge3 ACCESS p_DSSOT3MagSizeLarge;
	p_bSOTMagSizeLarge4 ACCESS p_DSSOT4MagSizeLarge;

	p_bDisableFMWarning ACCESS p_McParamDisableFMWarning;

	//For Siemen + We fab
	p_eCustomerReq ACCESS p_NtParamCustomerReq;

	p_bOpsMagConvLD1ReadRFID ACCESS p_OpsMagConvLD1ReadRFID;
	p_bOpsMagConvLD1WriteRFID ACCESS p_OpsMagConvLD1WriteRFID;

	p_bOpsMagConvLD2ReadRFID ACCESS p_OpsMagConvLD2ReadRFID;
	p_bOpsMagConvLD2WriteRFID ACCESS p_OpsMagConvLD2WriteRFID;

	p_bOpsMagConvLD3ReadRFID ACCESS p_OpsMagConvLD3ReadRFID;
	p_bOpsMagConvLD3WriteRFID ACCESS p_OpsMagConvLD3WriteRFID;

	(* Always Change If Project Change *)

END_ACTION
```

#### InputRef_Link.var - Change By Project
```iecst
(*2018-12-08*)
(**)
(*External Data*)
(**)
VAR
	p_bLinkCoverSWSig : REFERENCE TO BOOL;
	p_bLinkSafetyRlySig : REFERENCE TO BOOL;
	p_bLinkAlarmWarning : REFERENCE TO BOOL;
	p_bLinkAlarmInfo : REFERENCE TO BOOL;
	p_bLinkError : REFERENCE TO BOOL;
	p_eLinkLDMag : REFERENCE TO eLDMag;
	p_eLinkAGVComProtocol : REFERENCE TO eMcAGVCommProtocol;
END_VAR
```

#### Act_Link.st - Change By Project
```iecst
(** 2018-12-08 **)
ACTION Act_Link:

	tyDTMagToAGV.bEStopErr  := (p_bLinkCoverSWSig = FALSE) OR (p_bLinkSafetyRlySig = FALSE);

END_ACTION
```

#### Act_InitLocal.st - Do Not Change!!!
```iecst
(** 2019-01-20 **)
ACTION Act_InitLocal:

	//Input Reference Link To Local Variable
	p_udiRstErr ACCESS ADR(udiRstErr);
	p_bPrep ACCESS ADR(bPrep);
	p_bEn ACCESS ADR(bEn);
	p_bDis ACCESS ADR(bDis);
	p_sProgNm ACCESS ADR(sProgNm);
	p_bNtSettingsLoadDone ACCESS ADR(bNtSettingsLoadDone);
	p_tyDTMagToAGV1 ACCESS ADR(tyDTMagToAGV1);

END_ACTION
```

#### Act_Initial.st - Do Not Change!!!
```iecst
(** 2019-01-12 **)
ACTION Act_Initial:

	//Initial
	sStatTxt	:= a_sStatText[eStat];

	fbConnect(bEn := FALSE);
	fbGetNodeHdlListCrtSub(bEn := FALSE);
	fbGetNodeHdlListCrtSub.a_sServerTagNm[0] := '::AGV:tyTagFromLoader.tyTagStatOfPlatForms[1].usiMagBrdUnloadCnt';
	fbGetNodeHdlListCrtSub.a_sServerTagNm[1] := '::AGV:tyTagFromLoader.tyTagStatOfPlatForms[1].bFinishedLoading';
	fbGetNodeHdlListCrtSub.a_sServerTagNm[2] := '::AGV:tyTagFromLoader.tyTagStatOfPlatForms[2].usiMagBrdUnloadCnt';
	fbGetNodeHdlListCrtSub.a_sServerTagNm[3] := '::AGV:tyTagFromLoader.tyTagStatOfPlatForms[2].bFinishedLoading';
	fbGetNodeHdlListCrtSub.a_sServerTagNm[4] := '::AGV:tyTagFromLoader.tyTagStatOfPlatForms[3].usiMagBrdUnloadCnt';
	fbGetNodeHdlListCrtSub.a_sServerTagNm[5] := '::AGV:tyTagFromLoader.tyTagStatOfPlatForms[3].bFinishedLoading';
	fbGetNodeHdlListCrtSub.a_sServerTagNm[6] := '::AGV:tyTagFromLoader.tyTagStatOfPlatForms[4].usiMagBrdUnloadCnt';
	fbGetNodeHdlListCrtSub.a_sServerTagNm[7] := '::AGV:tyTagFromLoader.tyTagStatOfPlatForms[4].bFinishedLoading';

	fbCreateSub(bEn := FALSE);
	fbAddMoniteredList(bEn := FALSE);

	fbAddMoniteredList.a_sClientTagNm[0] := '::AGV:tyTagFromLoader.tyTagStatOfPlatForms[1].usiMagBrdUnloadCnt';
	fbAddMoniteredList.a_sClientTagNm[1] := '::AGV:tyTagFromLoader.tyTagStatOfPlatForms[1].bFinishedLoading';
	fbAddMoniteredList.a_sClientTagNm[2] := '::AGV:tyTagFromLoader.tyTagStatOfPlatForms[2].usiMagBrdUnloadCnt';
	fbAddMoniteredList.a_sClientTagNm[3] := '::AGV:tyTagFromLoader.tyTagStatOfPlatForms[2].bFinishedLoading';
	fbAddMoniteredList.a_sClientTagNm[4] := '::AGV:tyTagFromLoader.tyTagStatOfPlatForms[3].usiMagBrdUnloadCnt';
	fbAddMoniteredList.a_sClientTagNm[5] := '::AGV:tyTagFromLoader.tyTagStatOfPlatForms[3].bFinishedLoading';
	fbAddMoniteredList.a_sClientTagNm[6] := '::AGV:tyTagFromLoader.tyTagStatOfPlatForms[4].usiMagBrdUnloadCnt';
	fbAddMoniteredList.a_sClientTagNm[7] := '::AGV:tyTagFromLoader.tyTagStatOfPlatForms[4].bFinishedLoading';

	fbRmvMoniteredList(bEn := FALSE);

	fbDeleteSub(bEn := FALSE);
	fbDisconnect(bEn := FALSE);
END_ACTION
```

#### Act_Main.st - Do Not Change!!!
```iecst
(** 2019-01-20 **)
ACTION Act_Main:

	tyTagToMes.sMachineName := p_sJobNo;
	tyTagToMes.bError := p_bLinkError;
	tyTagToMes.bWarning := p_bLinkAlarmWarning OR p_bLinkAlarmInfo;

	bFleetManagerActive := p_bDIFleetManagerActive;

	CASE p_eLinkAGVComProtocol OF
		McSetAGVCommOPCUA, McSetAGVCommHardIO:
			fbFMOnTimeout(IN:= bFleetManagerActive);
			fbFMOffTimeout(IN:= bFleetManagerActive = FALSE);
			IF fbFMOnTimeout.Q OR fbFMOffTimeout.Q THEN
				IF p_bDisableFMWarning = FALSE THEN
					udiStatus1 := 10006;
				ELSE
					udiStatus1 := 0;
				END_IF
			ELSE
				udiStatus1 := 0;
			END_IF
		McSetAGVCommDisabled:
			udiStatus1 := 0;
	END_CASE

	CASE p_eLinkLDMag OF
		LDMagDual:
			tyTagToMes.nNumberOfPlatforms:= 2;

		LDMagTriple:
			tyTagToMes.nNumberOfPlatforms:= 3;

		LDMagQuadruple:
			tyTagToMes.nNumberOfPlatforms:= 4;
	END_CASE

	//Online Pulse Status- 500ms Pulse
	fbConnectionAGVTm(IN:= tyTagToMes.bActive = FALSE);
	IF fbConnectionAGVTm.Q THEN
		tyTagToMes.bActive := TRUE;
		//	bInternalAGVOnline := TRUE;
	END_IF

	fbConnectionAGVTm1(IN:= tyTagToMes.bActive);
	IF fbConnectionAGVTm1.Q THEN
		tyTagToMes.bActive := FALSE;
		//	bInternalAGVOnline := FALSE;
	END_IF

	//Simulation from HMI
	IF p_bUIAGVSimulationOn THEN
		bAGVOnline := p_bUIAGVOnline;

		tyAGVToDTMag.bVEHAuto := p_tyUIAGVToDTMagSimulateData.bVEHAuto;
		tyAGVToDTMag.bVEHInPos1 := p_tyUIAGVToDTMagSimulateData.bVEHInPos1;
		tyAGVToDTMag.bVEHInPos2 := p_tyUIAGVToDTMagSimulateData.bVEHInPos2;
		tyAGVToDTMag.bVEHInPos3 := p_tyUIAGVToDTMagSimulateData.bVEHInPos3;
		tyAGVToDTMag.bVEHInPos4 := p_tyUIAGVToDTMagSimulateData.bVEHInPos4;
		tyAGVToDTMag.bVEH1Occupied := p_tyUIAGVToDTMagSimulateData.bVEH1Occupied;
		tyAGVToDTMag.bVEH2Occupied := p_tyUIAGVToDTMagSimulateData.bVEH2Occupied;
		tyAGVToDTMag.bVEH3Occupied := p_tyUIAGVToDTMagSimulateData.bVEH3Occupied;
		tyAGVToDTMag.bVEH4Occupied := p_tyUIAGVToDTMagSimulateData.bVEH4Occupied;
		bInternalAGVSimulateOn := TRUE;

	END_IF

	IF EDGEPOS( p_bUIAGVSimulationOn = FALSE) THEN
		bAGVOnline := FALSE;

		tyAGVToDTMag.bVEHAuto := FALSE;
		tyAGVToDTMag.bVEHInPos1 := FALSE;
		tyAGVToDTMag.bVEHInPos2 := FALSE;
		tyAGVToDTMag.bVEHInPos3 := FALSE;
		tyAGVToDTMag.bVEHInPos4 := FALSE;
		tyAGVToDTMag.bVEH1Occupied := FALSE;
		tyAGVToDTMag.bVEH2Occupied := FALSE;
		tyAGVToDTMag.bVEH3Occupied := FALSE;
		tyAGVToDTMag.bVEH4Occupied := FALSE;
		bInternalAGVSimulateOn := FALSE;

	END_IF

	IF p_bOpsRun AND p_eLinkAGVComProtocol = McSetAGVCommOPCUA THEN
		bInternalAGVOnline := TRUE;
		tyTagToMes.bAuto_Run := TRUE;
		//Magazine Conveyor 1
		tyDTMagToAGV.bCI1Auto					:= p_tyDTMagToAGV1.bCI1Auto;
		tyDTMagToAGV.bCI1Rdy  					:= p_tyDTMagToAGV1.bCI1Rdy;
		tyDTMagToAGV.bCI1MagazineEmpty			:= p_tyDTMagToAGV1.bCI1MagazineEmpty;
		tyDTMagToAGV.bCI1Occupied				:= p_tyDTMagToAGV1.bCI1Occupied;
		tyDTMagToAGV.bCI1Running				:= p_tyDTMagToAGV1.bCI1Running;
		tyDTMagToAGV.bCI1IncorrectMagazineModel	:= p_bIncorrectMagazine1;

		tyTagToMes.tyTagStatOfPlatforms[1].bReqAIVToBring	:= p_bRequestToBring1;
		tyTagToMes.tyTagStatOfPlatforms[1].bReqAIVToGet		:= p_bRequestToGet1;
		tyTagToMes.tyTagStatOfPlatforms[1].bError			:= p_bSOTMagError1;
		tyTagToMes.tyTagStatOfPlatforms[1].bSizeLarge		:= p_bSOTMagSizeLarge1;
		tyTagToMes.tyTagStatOfPlatforms[1].bReady			:= p_bSOTMagReady1;
		tyTagToMes.tyTagStatOfPlatforms[1].bAvailable		:= p_bSOTMagAvailable1;

		//Magazine Conveyor 2
		tyDTMagToAGV.bCI2Auto					:= p_tyDTMagToAGV2.bCI2Auto;
		tyDTMagToAGV.bCI2Rdy  					:= p_tyDTMagToAGV2.bCI2Rdy;
		tyDTMagToAGV.bCI2MagazineEmpty			:= p_tyDTMagToAGV2.bCI2MagazineEmpty;
		tyDTMagToAGV.bCI2Occupied				:= p_tyDTMagToAGV2.bCI2Occupied;
		tyDTMagToAGV.bCI2Running				:= p_tyDTMagToAGV2.bCI2Running;
		tyDTMagToAGV.bCI2IncorrectMagazineModel	:= p_bIncorrectMagazine2;

		tyTagToMes.tyTagStatOfPlatforms[2].bReqAIVToBring	:= p_bRequestToBring2;
		tyTagToMes.tyTagStatOfPlatforms[2].bReqAIVToGet		:= p_bRequestToGet2;
		tyTagToMes.tyTagStatOfPlatforms[2].bError			:= p_bSOTMagError2;
		tyTagToMes.tyTagStatOfPlatforms[2].bSizeLarge		:= p_bSOTMagSizeLarge2;
		tyTagToMes.tyTagStatOfPlatforms[2].bReady			:= p_bSOTMagReady2;
		tyTagToMes.tyTagStatOfPlatforms[2].bAvailable		:= p_bSOTMagAvailable2;

		//Magazine Conveyor 3
		tyDTMagToAGV.bCI3Auto					:= p_tyDTMagToAGV3.bCI3Auto;
		tyDTMagToAGV.bCI3Rdy  					:= p_tyDTMagToAGV3.bCI3Rdy;
		tyDTMagToAGV.bCI3MagazineEmpty			:= p_tyDTMagToAGV3.bCI3MagazineEmpty;
		tyDTMagToAGV.bCI3Occupied				:= p_tyDTMagToAGV3.bCI3Occupied;
		tyDTMagToAGV.bCI3Running				:= p_tyDTMagToAGV3.bCI3Running;
		tyDTMagToAGV.bCI3IncorrectMagazineModel	:= p_bIncorrectMagazine3;

		tyTagToMes.tyTagStatOfPlatforms[3].bReqAIVToBring	:= p_bRequestToBring3;
		tyTagToMes.tyTagStatOfPlatforms[3].bReqAIVToGet		:= p_bRequestToGet3;
		tyTagToMes.tyTagStatOfPlatforms[3].bError			:= p_bSOTMagError3;
		tyTagToMes.tyTagStatOfPlatforms[3].bSizeLarge		:= p_bSOTMagSizeLarge3;
		tyTagToMes.tyTagStatOfPlatforms[3].bReady			:= p_bSOTMagReady3;
		tyTagToMes.tyTagStatOfPlatforms[3].bAvailable		:= p_bSOTMagAvailable3;

		//Magazine Conveyor 4
		tyDTMagToAGV.bCI4Auto					:= p_tyDTMagToAGV4.bCI4Auto;
		tyDTMagToAGV.bCI4Rdy  					:= p_tyDTMagToAGV4.bCI4Rdy;
		tyDTMagToAGV.bCI4MagazineEmpty			:= p_tyDTMagToAGV4.bCI4MagazineEmpty;
		tyDTMagToAGV.bCI4Occupied				:= p_tyDTMagToAGV4.bCI4Occupied;
		tyDTMagToAGV.bCI4Running				:= p_tyDTMagToAGV4.bCI4Running;
		tyDTMagToAGV.bCI4IncorrectMagazineModel	:= p_bIncorrectMagazine4;

		tyTagToMes.tyTagStatOfPlatforms[4].bReqAIVToBring	:= p_bRequestToBring4;
		tyTagToMes.tyTagStatOfPlatforms[4].bReqAIVToGet		:= p_bRequestToGet4;
		tyTagToMes.tyTagStatOfPlatforms[4].bError			:= p_bSOTMagError4;
		tyTagToMes.tyTagStatOfPlatforms[4].bSizeLarge		:= p_bSOTMagSizeLarge4;
		tyTagToMes.tyTagStatOfPlatforms[4].bReady			:= p_bSOTMagReady4;
		tyTagToMes.tyTagStatOfPlatforms[4].bAvailable		:= p_bSOTMagAvailable4;
		//To AGV Side to do Check Machine On

		bMachineOnline := TRUE;

		//Siemens + Wefabricate
		CASE p_eCustomerReq OF
			Siemens:
				tyTagToMes.tyTagStatOfPlatforms[1].bReadRFID 	:= p_bOpsMagConvLD1ReadRFID;
				tyTagToMes.tyTagStatOfPlatforms[1].bWriteRFID 	:= p_bOpsMagConvLD1WriteRFID;
				tyTagToMes.tyTagStatOfPlatforms[2].bReadRFID 	:= p_bOpsMagConvLD2ReadRFID;
				tyTagToMes.tyTagStatOfPlatforms[2].bWriteRFID 	:= p_bOpsMagConvLD2WriteRFID;
				tyTagToMes.tyTagStatOfPlatforms[3].bReadRFID 	:= p_bOpsMagConvLD3ReadRFID;
				tyTagToMes.tyTagStatOfPlatforms[3].bWriteRFID 	:= p_bOpsMagConvLD3WriteRFID;
			We_Fabricate:
				tyTagToMes.tyTagStatOfPlatforms[1].bMagLoaded 	:= p_bOpsMagConvLD1ReadRFID;
				tyTagToMes.tyTagStatOfPlatforms[2].bMagLoaded 	:= p_bOpsMagConvLD2ReadRFID;
				tyTagToMes.tyTagStatOfPlatforms[3].bMagLoaded 	:= p_bOpsMagConvLD3ReadRFID;
		END_CASE

	ELSE
		bInternalAGVOnline := FALSE;
		tyTagToMes.bAuto_Run := FALSE;
		//Magazine Conveyor 1
		tyDTMagToAGV.bCI1Auto					:= FALSE;
		tyDTMagToAGV.bCI1Rdy  					:= FALSE;
		tyDTMagToAGV.bCI1Running				:= FALSE;

		//Magazine Conveyor 2
		tyDTMagToAGV.bCI2Auto					:= FALSE;
		tyDTMagToAGV.bCI2Rdy  					:= FALSE;
		tyDTMagToAGV.bCI2Running				:= FALSE;

		//Magazine Conveyor 3
		tyDTMagToAGV.bCI3Auto					:= FALSE;
		tyDTMagToAGV.bCI3Rdy  					:= FALSE;
		tyDTMagToAGV.bCI3Running				:= FALSE;

		//Magazine Conveyor 4
		tyDTMagToAGV.bCI4Auto					:= FALSE;
		tyDTMagToAGV.bCI4Rdy  					:= FALSE;
		tyDTMagToAGV.bCI4Running				:= FALSE;

		bMachineOnline := FALSE;

		//Siemens
		tyTagToMes.tyTagStatOfPlatforms[1].bReadRFID 	:= FALSE;
		tyTagToMes.tyTagStatOfPlatforms[1].bWriteRFID 	:= FALSE;
		tyTagToMes.tyTagStatOfPlatforms[2].bReadRFID 	:= FALSE;
		tyTagToMes.tyTagStatOfPlatforms[2].bWriteRFID 	:= FALSE;
		tyTagToMes.tyTagStatOfPlatforms[3].bReadRFID 	:= FALSE;
		tyTagToMes.tyTagStatOfPlatforms[3].bWriteRFID 	:= FALSE;

		IF p_bManual THEN

			tyTagToMes.tyTagStatOfPlatforms[1].bReqAIVToBring	:= p_bUIRequestToBring1;
			tyTagToMes.tyTagStatOfPlatforms[1].bReqAIVToGet		:= p_bUIRequestToGet1;
			tyTagToMes.tyTagStatOfPlatforms[1].bError			:= p_bUISOTMagError1;
			tyTagToMes.tyTagStatOfPlatforms[1].bSizeLarge		:= p_bUISOTMagSizeLarge1;
			tyTagToMes.tyTagStatOfPlatforms[1].bReady			:= p_bUISOTMagReady1;
			tyTagToMes.tyTagStatOfPlatforms[1].bAvailable		:= p_bUISOTMagAvailable1;

			tyTagToMes.tyTagStatOfPlatforms[2].bReqAIVToBring	:= p_bUIRequestToBring2;
			tyTagToMes.tyTagStatOfPlatforms[2].bReqAIVToGet		:= p_bUIRequestToGet2;
			tyTagToMes.tyTagStatOfPlatforms[2].bError			:= p_bUISOTMagError2;
			tyTagToMes.tyTagStatOfPlatforms[2].bSizeLarge		:= p_bUISOTMagSizeLarge2;
			tyTagToMes.tyTagStatOfPlatforms[2].bReady			:= p_bUISOTMagReady2;
			tyTagToMes.tyTagStatOfPlatforms[2].bAvailable		:= p_bUISOTMagAvailable2;

			tyTagToMes.tyTagStatOfPlatforms[3].bReqAIVToBring	:= p_bUIRequestToBring3;
			tyTagToMes.tyTagStatOfPlatforms[3].bReqAIVToGet		:= p_bUIRequestToGet3;
			tyTagToMes.tyTagStatOfPlatforms[3].bError			:= p_bUISOTMagError3;
			tyTagToMes.tyTagStatOfPlatforms[3].bSizeLarge		:= p_bUISOTMagSizeLarge3;
			tyTagToMes.tyTagStatOfPlatforms[3].bReady			:= p_bUISOTMagReady3;
			tyTagToMes.tyTagStatOfPlatforms[3].bAvailable		:= p_bUISOTMagAvailable3;

			tyTagToMes.tyTagStatOfPlatforms[4].bReqAIVToBring	:= p_bUIRequestToBring4;
			tyTagToMes.tyTagStatOfPlatforms[4].bReqAIVToGet		:= p_bUIRequestToGet4;
			tyTagToMes.tyTagStatOfPlatforms[4].bError			:= p_bUISOTMagError4;
			tyTagToMes.tyTagStatOfPlatforms[4].bSizeLarge		:= p_bUISOTMagSizeLarge4;
			tyTagToMes.tyTagStatOfPlatforms[4].bReady			:= p_bUISOTMagReady4;
			tyTagToMes.tyTagStatOfPlatforms[4].bAvailable		:= p_bUISOTMagAvailable4;

		ELSE

			tyTagToMes.tyTagStatOfPlatforms[1].bReqAIVToBring	:= FALSE;
			tyTagToMes.tyTagStatOfPlatforms[1].bReqAIVToGet		:= FALSE;
			tyTagToMes.tyTagStatOfPlatforms[1].bError			:= FALSE;
			tyTagToMes.tyTagStatOfPlatforms[1].bSizeLarge		:= FALSE;
			tyTagToMes.tyTagStatOfPlatforms[1].bReady			:= FALSE;
			tyTagToMes.tyTagStatOfPlatforms[1].bAvailable		:= FALSE;

			tyTagToMes.tyTagStatOfPlatforms[2].bReqAIVToBring	:= FALSE;
			tyTagToMes.tyTagStatOfPlatforms[2].bReqAIVToGet		:= FALSE;
			tyTagToMes.tyTagStatOfPlatforms[2].bError			:= FALSE;
			tyTagToMes.tyTagStatOfPlatforms[2].bSizeLarge		:= FALSE;
			tyTagToMes.tyTagStatOfPlatforms[2].bReady			:= FALSE;
			tyTagToMes.tyTagStatOfPlatforms[2].bAvailable		:= FALSE;

			tyTagToMes.tyTagStatOfPlatforms[3].bReqAIVToBring	:= FALSE;
			tyTagToMes.tyTagStatOfPlatforms[3].bReqAIVToGet		:= FALSE;
			tyTagToMes.tyTagStatOfPlatforms[3].bError			:= FALSE;
			tyTagToMes.tyTagStatOfPlatforms[3].bSizeLarge		:= FALSE;
			tyTagToMes.tyTagStatOfPlatforms[3].bReady			:= FALSE;
			tyTagToMes.tyTagStatOfPlatforms[3].bAvailable		:= FALSE;

			tyTagToMes.tyTagStatOfPlatforms[4].bReqAIVToBring	:= FALSE;
			tyTagToMes.tyTagStatOfPlatforms[4].bReqAIVToGet		:= FALSE;
			tyTagToMes.tyTagStatOfPlatforms[4].bError			:= FALSE;
			tyTagToMes.tyTagStatOfPlatforms[4].bSizeLarge		:= FALSE;
			tyTagToMes.tyTagStatOfPlatforms[4].bReady			:= FALSE;
			tyTagToMes.tyTagStatOfPlatforms[4].bAvailable		:= FALSE;

		END_IF

	END_IF

END_ACTION
```

#### Act_Background.st - Do Not Change!!!
```iecst
(** 2023-09-23 **)
ACTION Act_Background:
	//for OPCUA Loader Connect to Unloader AGV solution
	IF NOT(bTest) THEN

		fbConnect(bEn := FALSE);
		fbGetNodeHdlListCrtSub(bEn := FALSE);
		fbCreateSub(bEn := FALSE);
		fbAddMoniteredList(bEn := FALSE);
		fbRmvMoniteredList(bEn := FALSE);
		fbDeleteSub(bEn := FALSE);
		fbDisconnect(bEn := FALSE);
	ELSE
		CASE usiStep OF
			0:
				//Connect HMI OPCUA Server
				fbConnect.tyOPCUAParam.sIPAddr	:= '192.168.0.20';
				fbConnect.tyOPCUAParam.sPort := '4840';
				fbConnect(bEn := TRUE);

				IF fbConnect.udiStatus = 0 THEN
					dwConnectionHdl	:= fbConnect.dwConnectionHdl;
					fbConnect(bEn := FALSE);

				//	bConnected := TRUE;

					usiStep	:= 1;
				ELSIF fbConnect.udiStatus < 65534 THEN
					fbConnect(bEn := FALSE);

				//	bConnected := FALSE;
					usiStep := 0;
				END_IF

			1:
				//Node Handle List Read

				fbGetNodeHdlListCrtSub.usiNSIdx := 6;
				fbGetNodeHdlListCrtSub.uiTagNmCnt := 8;	 //tyTagFromLoader.tyTagStatOfPlatForms[1].bFinishedLoading

				fbGetNodeHdlListCrtSub.dwConnectionHdl := dwConnectionHdl;
				fbGetNodeHdlListCrtSub(bEn := TRUE);

				IF fbGetNodeHdlListCrtSub.udiStatus = 0 THEN
					tyPubSubHdls.a_dwHdls := fbGetNodeHdlListCrtSub.a_dwNodeHdlList;
					fbGetNodeHdlListCrtSub(bEn := FALSE);

					usiStep := 2;
				ELSIF fbGetNodeHdlListCrtSub.udiStatus < 65534 THEN
					fbGetNodeHdlListCrtSub(bEn := FALSE);

					usiStep := 9;
				END_IF

			2:
				//Create Sub
				fbCreateSub.dwConnectionHdl := dwConnectionHdl;
				fbCreateSub.bPublishingEn := TRUE;
				fbCreateSub.bytePriority := 0;

				fbCreateSub(bEn := TRUE,tPublishingInterval := T#1s);

				IF fbCreateSub.udiStatus = 0 THEN
					dwSubHdl := fbCreateSub.dwSubHdl;
					fbCreateSub(bEn := FALSE);

					usiStep := 3;

				ELSIF fbCreateSub.udiStatus < 65534 THEN
					fbCreateSub(bEn := FALSE);

					usiStep := 9;
				END_IF

			3:
				//Add Monitor Item List
				eStatus := Busy;

				fbAddMoniteredList.dwSubHdl := dwSubHdl;
				fbAddMoniteredList.a_dwNodeHdlList := tyPubSubHdls.a_dwHdls;

				fbAddMoniteredList.uiTagNmCount := 8;

				fbAddMoniteredList(bEn := TRUE);

				IF fbAddMoniteredList.udiStatus = 0 THEN
					a_dwMonitoringHdl := fbAddMoniteredList.a_dwMonitorHdl;
					//a_bValueChange to be added
					//fbAddMoniteredList(bEn := FALSE);
					usiStep := 99;
					fbAddMoniteredList(bEn:= FALSE);
					//usiChkIpAddrStep := 4;
				ELSIF fbAddMoniteredList.udiStatus < 65534 THEN
					fbAddMoniteredList(bEn := FALSE);

					usiStep := 9;
				END_IF
			99:
//				IF NOT(bDisconnect) THEN
//					fbAddMoniteredList;
//				ELSE
//					fbAddMoniteredList(bEn:= FALSE);
//				END_IF
			4:
			//Remove Item List
			fbRmvMoniteredList.dwSubHdl := dwSubHdl;
			fbRmvMoniteredList.uiTagNmCount := 8;
			fbRmvMoniteredList.a_dwMonitorHld:= a_dwMonitoringHdl;
			fbRmvMoniteredList(bEn := TRUE);

			IF fbRmvMoniteredList.udiStatus = 0 THEN

				fbRmvMoniteredList(bEn := FALSE);
				//uiTagNmCount := 0;
				//memset(ADR(a_dwMonitoringHdl),0,SIZEOF(a_dwMonitoringHdl));

				usiStep := 99;
			ELSIF fbRmvMoniteredList.udiStatus < 65534 THEN
				fbRmvMoniteredList(bEn := FALSE);

			//	usiStep := 9;
			END_IF

		5:
			//Delete Subscription
			fbDeleteSub.dwSubHdl := dwSubHdl;
			fbDeleteSub(bEn := TRUE);

			IF fbDeleteSub.udiStatus = 0 THEN
				//dwSubHdl := 0;
				fbDeleteSub(bEn := FALSE);

				usiStep := 99;
			ELSIF fbDeleteSub.udiStatus < 65534 THEN
				fbDeleteSub(bEn := FALSE);

			//	usiStep := 9;
			END_IF

		6:
				//Release Node
				fbRlsNodeHdlList.a_dwNodeHdlList := tyPubSubHdls.a_dwHdls;
				fbRlsNodeHdlList.uiTagNmCnt := 8;
				fbRlsNodeHdlList.dwConnectionHdl := dwConnectionHdl;
				fbRlsNodeHdlList(bEn := TRUE);

				IF fbRlsNodeHdlList.udiStatus = 0 THEN

				//	memset(ADR(tyPubSubHdls.a_dwHdls),0,SIZEOF(tyPubSubHdls.a_dwHdls));
					fbRlsNodeHdlList(bEn := FALSE);
					usiStep := 99;
				ELSIF fbRlsNodeHdlList.udiStatus < 65534 THEN
					fbRlsNodeHdlList(bEn := FALSE);

					//	usiStep := 9;
				END_IF

		9:
			//Disconnect
			fbDisconnect.dwConnectionHdl		:= dwConnectionHdl;
			fbDisconnect(bEn := TRUE);

			IF fbDisconnect.udiStatus = 0 THEN
				fbDisconnect(bEn := FALSE);
				memset(ADR(tyPubSubHdls.a_dwHdls),0,SIZEOF(tyPubSubHdls.a_dwHdls));
				memset(ADR(a_dwMonitoringHdl),0,SIZEOF(a_dwMonitoringHdl));
				dwConnectionHdl	:= 0;
				dwSubHdl		:= 0;

				bTest := FALSE;
				eStatus := Done;

				//usiStep	:=0;

			ELSIF fbDisconnect.udiStatus < 65534 THEN
				fbDisconnect(bEn := FALSE);
				dwConnectionHdl := 0;
			//	bConnected := FALSE;
				udiStatus			:= 10013; //Failed to Call Load Configuration Method

				//usiStep := 0;
			END_IF

		END_CASE

	END_IF

END_ACTION
```

#### Act_Alarm.st - Do Not Change!!!
```iecst
(** 2019-03-25 **)
ACTION Act_Alarm:

	//Error
	IF EDGEPOS(eStatus = Error) THEN

		tyAlmData.sProgNm		:= p_sProgNm;
		tyAlmData.udiCode		:= udiStatus;
		tyAlmData.eSeverity		:= AlmSeverityError;
		tyAlmData.udiRunTime	:= tyAlmData.udiRunTime + 1;
		tyAlmData.bAlm			:= TRUE;
		tyAlmData.udiModuleNum  := udiModuleNum;
		g_sAGVComProgNm		:= p_sProgNm;
		//Get Error Message
		IF tyAlmData.udiCode < 10000 OR tyAlmData.udiCode > 10099 THEN
			tyAlmData.sAlmMsg	:= 'Unknown';
			tyAlmData.sRcyMsg	:= 'Unknown';
		ELSE
			tyAlmData.sAlmMsg	:= a_tyAlmText[tyAlmData.udiCode].sAlmText;
			tyAlmData.sRcyMsg	:= a_tyAlmText[tyAlmData.udiCode].sRcyText;
		END_IF

		sStatTxt	:= tyAlmData.sAlmMsg;

	ELSIF bRstErr AND (tyAlmData.udiCode <> 0) THEN

		tyAlmData.udiCode	:= 0;
		tyAlmData.eSeverity	:= AlmSeverityNA;
		tyAlmData.sAlmMsg	:= '';
		tyAlmData.sRcyMsg	:= '';
		tyAlmData.bAlm			:= FALSE;
		sStatTxt	:= a_sStatText[eStat];

	END_IF

END_ACTION
```

#### Act_Alarm1.st - Do Not Change!!!
```iecst
(** 2019-03-25 **)
ACTION Act_Alarm1:

		tyAlmData1.sProgNm		:= p_sProgNm;
		tyAlmData1.udiCode		:= udiStatus1;
		tyAlmData1.eSeverity	:= AlmSeverityWarning;
		tyAlmData1.udiRunTime	:= tyAlmData1.udiRunTime + 1;
		tyAlmData1.bWarning		:= TRUE;
		tyAlmData1.udiModuleNum  := udiModuleNum;
		g_sAGVComProgNm			:= p_sProgNm;
		//Get Error Message
		IF tyAlmData1.udiCode < 10000 OR tyAlmData1.udiCode > 10099 THEN
			tyAlmData1.sAlmMsg	:= 'Unknown';
			tyAlmData1.sRcyMsg	:= 'Unknown';
		ELSE
			tyAlmData1.sAlmMsg	:= a_tyAlmText[tyAlmData1.udiCode].sAlmText;
			tyAlmData1.sRcyMsg	:= a_tyAlmText[tyAlmData1.udiCode].sRcyText;
		END_IF

END_ACTION
```

#### InputRef.var - Do Not Change!!!
```iecst
(*2019-01-20*)
(**)
(*General*)
VAR
	p_udiRstErr : REFERENCE TO UDINT;
	p_bPrep : REFERENCE TO BOOL;
	p_bEn : REFERENCE TO BOOL;
	p_bDis : REFERENCE TO BOOL;
END_VAR
(**)
(*Configuration*)
VAR
	p_sProgNm : REFERENCE TO STRING[15];
	p_bNtSettingsLoadDone : REFERENCE TO BOOL;
	p_sJobNo : REFERENCE TO STRING[30];
END_VAR
(**)
(*Input*)
VAR
	p_bManual : REFERENCE TO BOOL;
	p_tyDTMagToAGV1 : REFERENCE TO tyTagDTMagToAGV;
	p_tyDTMagToAGV2 : REFERENCE TO tyTagDTMagToAGV;
	p_tyDTMagToAGV3 : REFERENCE TO tyTagDTMagToAGV;
	p_tyDTMagToAGV4 : REFERENCE TO tyTagDTMagToAGV;
	p_bOpsRun : REFERENCE TO BOOL;
	p_bLinkOpsSimu : REFERENCE TO BOOL;
	p_bIncorrectMagazine1 : REFERENCE TO BOOL;
	p_bIncorrectMagazine2 : REFERENCE TO BOOL;
	p_bIncorrectMagazine3 : REFERENCE TO BOOL;
	p_bIncorrectMagazine4 : REFERENCE TO BOOL;
END_VAR
(*Simulate Data*)
VAR
	p_tyUIAGVToDTMagSimulateData : REFERENCE TO tyTagAGVToDTMag;
	p_bUIAGVOnline : REFERENCE TO BOOL;
	p_bUIAGVSimulationOn : REFERENCE TO BOOL;
	p_bAGVRdyEnter1 : REFERENCE TO BOOL;
	p_bAGVRdyExit1 : REFERENCE TO BOOL;
	p_bAGVRdyEnter2 : REFERENCE TO BOOL;
	p_bAGVRdyExit2 : REFERENCE TO BOOL;
	p_bAGVRdyEnter3 : REFERENCE TO BOOL;
	p_bAGVRdyExit3 : REFERENCE TO BOOL;
	p_bAGVRdyEnter4 : REFERENCE TO BOOL;
	p_bAGVRdyExit4 : REFERENCE TO BOOL;
END_VAR
(**)
VAR
	p_bRequestToBring1 : REFERENCE TO BOOL;
	p_bRequestToBring2 : REFERENCE TO BOOL;
	p_bRequestToBring3 : REFERENCE TO BOOL;
	p_bRequestToBring4 : REFERENCE TO BOOL;
	p_bRequestToGet1 : REFERENCE TO BOOL;
	p_bRequestToGet2 : REFERENCE TO BOOL;
	p_bRequestToGet3 : REFERENCE TO BOOL;
	p_bRequestToGet4 : REFERENCE TO BOOL;
END_VAR
(**)
VAR
	p_bDIFleetManagerActive : REFERENCE TO BOOL;
	p_bUISOTMagError1 : REFERENCE TO BOOL;
	p_bUISOTMagError2 : REFERENCE TO BOOL;
	p_bUISOTMagError3 : REFERENCE TO BOOL;
	p_bUISOTMagError4 : REFERENCE TO BOOL;
	p_bUISOTMagReady1 : REFERENCE TO BOOL;
	p_bUISOTMagReady2 : REFERENCE TO BOOL;
	p_bUISOTMagReady3 : REFERENCE TO BOOL;
	p_bUISOTMagReady4 : REFERENCE TO BOOL;
	p_bUISOTMagAvailable1 : REFERENCE TO BOOL;
	p_bUISOTMagAvailable2 : REFERENCE TO BOOL;
	p_bUISOTMagAvailable3 : REFERENCE TO BOOL;
	p_bUISOTMagAvailable4 : REFERENCE TO BOOL;
	p_bUISOTMagSizeLarge1 : REFERENCE TO BOOL;
	p_bUISOTMagSizeLarge2 : REFERENCE TO BOOL;
	p_bUISOTMagSizeLarge3 : REFERENCE TO BOOL;
	p_bUISOTMagSizeLarge4 : REFERENCE TO BOOL;
	p_bUIRequestToBring1 : REFERENCE TO BOOL;
	p_bUIRequestToBring2 : REFERENCE TO BOOL;
	p_bUIRequestToBring3 : REFERENCE TO BOOL;
	p_bUIRequestToBring4 : REFERENCE TO BOOL;
	p_bUIRequestToGet1 : REFERENCE TO BOOL;
	p_bUIRequestToGet2 : REFERENCE TO BOOL;
	p_bUIRequestToGet3 : REFERENCE TO BOOL;
	p_bUIRequestToGet4 : REFERENCE TO BOOL;
	p_bSOTMagError1 : REFERENCE TO BOOL;
	p_bSOTMagSizeLarge1 : REFERENCE TO BOOL;
	p_bSOTMagReady1 : REFERENCE TO BOOL;
	p_bSOTMagAvailable1 : REFERENCE TO BOOL;
	p_bSOTMagError2 : REFERENCE TO BOOL;
	p_bSOTMagSizeLarge2 : REFERENCE TO BOOL;
	p_bSOTMagReady2 : REFERENCE TO BOOL;
	p_bSOTMagAvailable2 : REFERENCE TO BOOL;
	p_bSOTMagError3 : REFERENCE TO BOOL;
	p_bSOTMagSizeLarge3 : REFERENCE TO BOOL;
	p_bSOTMagReady3 : REFERENCE TO BOOL;
	p_bSOTMagAvailable3 : REFERENCE TO BOOL;
	p_bSOTMagError4 : REFERENCE TO BOOL;
	p_bSOTMagSizeLarge4 : REFERENCE TO BOOL;
	p_bSOTMagReady4 : REFERENCE TO BOOL;
	p_bSOTMagAvailable4 : REFERENCE TO BOOL;
	p_eAGVComProtocol : REFERENCE TO eMcAGVCommProtocol;
	p_bDisableFMWarning : REFERENCE TO BOOL;
END_VAR
(*Simens*)
VAR
	p_eCustomerReq : REFERENCE TO eCustomer;
	p_bOpsMagConvLD1ReadRFID : REFERENCE TO BOOL;
	p_bOpsMagConvLD1WriteRFID : REFERENCE TO BOOL;
	p_bOpsMagConvLD2ReadRFID : REFERENCE TO BOOL;
	p_bOpsMagConvLD2WriteRFID : REFERENCE TO BOOL;
	p_bOpsMagConvLD3ReadRFID : REFERENCE TO BOOL;
	p_bOpsMagConvLD3WriteRFID : REFERENCE TO BOOL;
END_VAR
```

#### Local.var - Do Not Change!!!
```iecst
(*2019-01-20*)
(**)
(*Local Action, State & Status*)
VAR
	eAct : eAGVMagAction := AGVMagActIdle;
	eStat : eAGVMagAction := AGVMagActIdle;
	eStatus : eFBStatus := Idle;
	eStatus1 : eFBStatus := Idle;
	udiStatus : UDINT := 0;
	udiStatus1 : UDINT := 0;
	sStatTxt : STRING[100] := '';
	a_sStatText : ARRAY[0..50] OF STRING[100] := ['Idling','AGV Magazine Ready Enter And Communicating AGV','AGV Magazine Ready Exit And Communicating AGV',48('')];
END_VAR
(**)
(*Local Alarm*)
VAR
	tyAlmData : tyAlmDat;
	tyAlmData1 : tyAlmDat;
	a_tyAlmText : ARRAY[10000..10099] OF tyAlmTxt := [(sAlmText:='Magazine Is Present Before Entering',sRcyText:='Remove Magazine To Continue Operation.'),(sAlmText:='AGV Not In Enter Position',sRcyText:='Adjust AGV Position And Restart Operation.'),(sAlmText:='Transfer In Time Out While Transporting',sRcyText:='Adjust Magazine Position Or Transporting Time.'),(sAlmText:='Magazine Is Not Present Before Exiting',sRcyText:='Magazine Has Taken Away, Restart Operation.'),(sAlmText:='AGV Not In Exit Position',sRcyText:='Adjust AGV Position And Restart Operation.'),(sAlmText:='Transfer Out Time Out While Transporting',sRcyText:='Adjust Magazine Position Or Transporting Time.'),(sAlmText:='Fleet Manager Is Offline',sRcyText:='Please check the connectivity signal to Fleetmanger'),93((0))];
END_VAR
(**)
(*Local Output*)
VAR
	bMcRunRdy : BOOL;
	bRdyEnt : BOOL;
	bRdyExit : BOOL;
	bMag1Ent : BOOL;
	bMag1Exit : BOOL;
END_VAR
(**)
(*Local Input*)
VAR
	udiRstErr : UDINT := 0;
	bPrep : BOOL := TRUE;
	bEn : BOOL := TRUE;
	bDis : BOOL := FALSE;
	sProgNm : STRING[15] := 'AGVMag';
	bNtSettingsLoadDone : BOOL := TRUE;
	tyAGVToDTMag : tyTagAGVToDTMag;
	tyDTMagToAGV : tyTagDTMagToAGV;
	bAGVOnline : BOOL;
	bMachineOnline : BOOL;
	bInternalAGVOnline : BOOL;
	bFleetManagerActive : BOOL;
	fbFMOnTimeout : TON := (PT:=T#20s);
	fbFMOffTimeout : TON := (PT:=T#20s);
	bInternalAGVSimulateOn : BOOL;
	tyDTMagToAGV1 : tyTagDTMagToAGV;
	tyDTMagToAGV2 : tyTagDTMagToAGV;
	tyDTMagToAGV3 : tyTagDTMagToAGV;
	tyDTMagToAGV4 : tyTagDTMagToAGV;
END_VAR
(**)
(*Local*)
VAR
	bRstErr : BOOL;
	udiRstErrOld : UDINT;
	bInitDone : BOOL;
	bInitialDone : BOOL;
	usiStep : USINT;
	eStatOld : eAGVMagAction := AGVMagActIdle;
	fbConnectionTmCCS : TON := (PT:=T#250ms);
	fbConnectionAGVTm : TON := (PT:=T#250ms);
	fbConnectionAGVTm1 : TON := (PT:=T#500ms);
END_VAR
(**)
VAR
	tyTagToMes : tyStatToMES;
	tyTagFromMes : tyStatFromMES;
	udiModuleNum : UDINT := 6111;
END_VAR
```

### Program Logical/AGVCom/AGV1 (IEC) - 1.00.0 - NtSMEMA v5.00.0

#### InputRef_Link.var
```iecst
(*2018-12-08*)
(**)
(*External Data*)
VAR
	p_bLinkAGVOnline : REFERENCE TO BOOL;
	p_bLinkOpsRun : REFERENCE TO BOOL;
END_VAR
(**)
VAR
	p_tyLinkBufferStat : REFERENCE TO tyBffrStat;
	p_tyLinkAGVtoDTMag : REFERENCE TO tyTagAGVToDTMag;
END_VAR
```

#### Local.var
```iecst
(*2019-01-20*)
(**)
(*Local Action, State & Status*)
VAR
	eAct : eAGVMagAction := AGVMagActIdle;
	eStat : eAGVMagAction := AGVMagActIdle;
	eStatus : eFBStatus := Idle;
	udiStatus : UDINT := 0;
	sStatTxt : STRING[100] := '';
	a_sStatText : ARRAY[0..50] OF STRING[100] := ['Idling','AGV Magazine Ready Enter And Communicating AGV','AGV Magazine Ready Exit And Communicating AGV',48('')];
END_VAR
(**)
(*Local Alarm*)
VAR
	tyAlmData : tyAlmDat;
	a_tyAlmText : ARRAY[10000..10099] OF tyAlmTxt := [(sAlmText:='Magazine Is Present Before Entering',sRcyText:='Remove Magazine To Continue Operation.'),(sAlmText:='AGV Not In Enter Position',sRcyText:='Adjust AGV Position And Restart Operation.'),(sAlmText:='Transfer In Time Out While Transporting',sRcyText:='Adjust Magazine Position Or Transporting Time Or Check Online Connection'),(sAlmText:='Magazine Is Not Present Before Exiting',sRcyText:='Magazine Has Taken Away, Restart Operation.'),(sAlmText:='AGV Not In Exit Position',sRcyText:='Adjust AGV Position And Restart Operation.'),(sAlmText:='Transfer Out Time Out While Transporting',sRcyText:='Adjust Magazine Position Or Transporting Time.'),(sAlmText:='AGV is not in Auto',sRcyText:='Make Sure AGV is in Auto'),(sAlmText:='Magazine is not Present in AGV while Entering',sRcyText:='Check AGV'),(sAlmText:='Magazine is Present in AGV while Exiting',sRcyText:='Check AGV'),(sAlmText:='AGV In Position Sensor is off while received the AGV in position signal',sRcyText:='Check AGV in position sensor'),(sAlmText:='SOT Error Signal Has Been Activated',sRcyText:='AIV Activated The Error Signal During Magazine Transportation'),0,88((0))];
END_VAR
(**)
(*Local Output*)
VAR
	bMcRunRdy : BOOL;
	bRdyEnt : BOOL;
	bRdyExit : BOOL;
	bMagEnt : BOOL;
	bMagExit : BOOL;
END_VAR
(**)
(*Local Input*)
VAR
	udiRstErr : UDINT := 0;
	bPrep : BOOL := TRUE;
	bEn : BOOL := TRUE;
	bDis : BOOL := FALSE;
	sProgNm : STRING[15] := 'AGVMag';
	bNtSettingsLoadDone : BOOL := TRUE;
	diTxInTimeOut : DINT;
	diTxOutTimeOut : DINT;
	eDirection : eConvDir;
	bBufferMagPresent : BOOL;
	bAGVInSen1 : BOOL;
	bAGVInSen2 : BOOL;
	bNtParamAGVInPosSenPrep : BOOL;
	bMagConvLftSen : BOOL;
	bMagConvRgtSen : BOOL;
	bMagConvMtrIn : BOOL;
	bMagConvMtrOut : BOOL;
	tyAGVToDTMag : tyTagAGVToDTMag;
	tyDTMagToAGV : tyTagDTMagToAGV;
END_VAR
(**)
(*Local*)
VAR
	bRstErr : BOOL;
	udiRstErrOld : UDINT;
	bInitDone : BOOL;
	bInitialDone : BOOL;
	usiStep : USINT;
	bEndSen : BOOL;
	bAGVInPosSen : BOOL;
	fbMagEmptyTm : TON := (PT:=T#2s);
	fbInPosErrTimer : TON;
	fbTxInTimer : TON;
	fbTxOutTimer : TON;
	fbMagOutTrig : F_TRIG;
	eStatOld : eAGVMagAction := AGVMagActIdle;
	fbCheckErrorTim : TON := (PT:=T#1s);
	bMagConvRun : BOOL;
	bMagConvRdy : BOOL;
	bMagConvAuto : BOOL;
	bMagConvOccupied : BOOL;
	bAIVOccupied : BOOL;
	bAIVAuto : BOOL;
	bAIVInPos : BOOL;
	udiModuleNum : UDINT := 6161;
END_VAR
```

#### Act_Alarm.st
```iecst
(** 2019-03-25 **)
ACTION Act_Alarm:

	//Error
	IF EDGEPOS(eStatus = Error) THEN

		tyAlmData.sProgNm		:= p_sProgNm;
		tyAlmData.udiCode		:= udiStatus;
		tyAlmData.eSeverity		:= AlmSeverityError;
		tyAlmData.udiRunTime	:= tyAlmData.udiRunTime + 1;
		tyAlmData.bAlm			:= TRUE;
		tyAlmData.udiModuleNum  := udiModuleNum;
		g_sAGVProgNm		:= p_sProgNm;
		//Get Error Message
		IF tyAlmData.udiCode < 10000 OR tyAlmData.udiCode > 10099 THEN
			tyAlmData.sAlmMsg	:= 'Unknown';
			tyAlmData.sRcyMsg	:= 'Unknown';
		ELSE
			tyAlmData.sAlmMsg	:= a_tyAlmText[tyAlmData.udiCode].sAlmText;
			tyAlmData.sRcyMsg	:= a_tyAlmText[tyAlmData.udiCode].sRcyText;
		END_IF

		sStatTxt	:= tyAlmData.sAlmMsg;

	ELSIF bRstErr AND (tyAlmData.udiCode <> 0) THEN

		tyAlmData.udiCode	:= 0;
		tyAlmData.eSeverity	:= AlmSeverityNA;
		tyAlmData.sAlmMsg	:= '';
		tyAlmData.sRcyMsg	:= '';
		tyAlmData.bAlm			:= FALSE;
		sStatTxt	:= a_sStatText[eStat];

	END_IF

END_ACTION
```

#### Act_InitGlobal.st
```iecst
(** 2018-12-08 **)
ACTION Act_InitGlobal:

	(* Always Change If Project Change *)

	//Pass Data To Link
	p_bLinkOpsRun ACCESS p_OpsRun;

	p_tyLinkBufferStat ACCESS p_Buffer1BffrStat;
	p_bLinkAGVOnline ACCESS p_AGVOnline;
	p_tyLinkAGVtoDTMag ACCESS p_AGVTagAGVToDTMag;

	//Pass Data To Internal Use
	p_eAct ACCESS p_OpsMagConvLD1AGVMagAct;
	p_udiRstErr	ACCESS p_RstErrReset;
	p_bPrep ACCESS p_NtParamProjAGVPrep;
	p_sProgNm ACCESS p_NtParamAGVMag1ProgNm;
	p_diTxInTimeOut ACCESS p_McParamMag1ConvRunTmOut;
	p_diTxOutTimeOut ACCESS p_McParamMag1ConvRunTmOut;
	p_eDirection ACCESS p_NtParamProjMagConvDir;
	p_bBufferMagPresent ACCESS p_DIMagPresentSen1;
	p_bMagConvLftSen ACCESS p_DIMagConvEntSen1;
	p_bMagConvRgtSen ACCESS p_DIMagPresentSen1;
	p_bMagConvMtrIn ACCESS p_MagConv2Clp1MtrSigOnOrLToR;
	p_bMagConvMtrOut ACCESS p_MagConv2Clp1MtrDirOrRToL;
	p_bNtSettingsLoadDone ACCESS p_StartupNtSettingsLoadDone;
	p_bAGVInPosSen1	ACCESS p_DIMag1AGVInPosSen1;
	p_bAGVInPosSen2	ACCESS p_DIMag1AGVInPosSen2;
	p_bNtParamAGVInPosSenPrep ACCESS p_NtParamProjAGVInPosSenPrep;
	p_bSOTRcvOk ACCESS p_DISOT1Receive;
	p_bSOTErr ACCESS p_DISOT1Error;
	p_bSOTRdy ACCESS p_DISOT1Ready;
	p_bSOTAvailable ACCESS p_DISOT1Available;
	p_bEn ACCESS p_McParamAGVComEn;

	(* Always Change If Project Change *)

END_ACTION
```

#### Act_Link.st
```iecst
(** 2018-12-08 **)
ACTION Act_Link:

	//Machine --> AGV ---> Communication On & Machine itself RUN Mode
	IF p_bLinkOpsRun = TRUE THEN

		tyDTMagToAGV.bCI1Auto := TRUE;
	ELSE
		tyDTMagToAGV.bCI1Auto	:= FALSE;
	END_IF

	tyDTMagToAGV.bCI1Occupied 			:= p_bBufferMagPresent OR p_bMagConvLftSen OR p_bMagConvRgtSen ;

	fbMagEmptyTm(IN:= p_bMagConvLftSen = FALSE AND p_bBufferMagPresent = FALSE);
	IF p_bBufferMagPresent AND p_tyLinkBufferStat.bBffrMty THEN
		tyDTMagToAGV.bCI1MagazineEmpty		:=  TRUE;
	ELSIF fbMagEmptyTm.Q THEN
		tyDTMagToAGV.bCI1MagazineEmpty		:=  FALSE;
	END_IF

	IF p_bLinkAGVOnline THEN

		p_tyAGVToDTMag.bVEHAuto		:= p_tyLinkAGVtoDTMag.bVEHAuto;
		p_tyAGVToDTMag.bVEHInPos1	:= p_tyLinkAGVtoDTMag.bVEHInPos1 AND bAGVInPosSen;
		p_tyAGVToDTMag.bVEHInPos2 	:= p_tyLinkAGVtoDTMag.bVEHInPos2;
		p_tyAGVToDTMag.bVEHInPos3 	:= p_tyLinkAGVtoDTMag.bVEHInPos3;
		p_tyAGVToDTMag.bVEH1Occupied	:= p_tyLinkAGVtoDTMag.bVEH1Occupied;
		p_tyAGVToDTMag.bVEH2Occupied	:= p_tyLinkAGVtoDTMag.bVEH2Occupied;
		p_tyAGVToDTMag.bVEH3Occupied	:= p_tyLinkAGVtoDTMag.bVEH3Occupied;
		p_tyAGVToDTMag.bVEHRunning	:= p_tyLinkAGVtoDTMag.bVEHRunning;

	ELSE

		p_tyAGVToDTMag.bVEHAuto		:= FALSE;
		p_tyAGVToDTMag.bVEHInPos1	:= FALSE;
		p_tyAGVToDTMag.bVEHInPos2 	:= FALSE;
		p_tyAGVToDTMag.bVEHInPos3 	:= FALSE;
		p_tyAGVToDTMag.bVEH1Occupied:= FALSE;
		p_tyAGVToDTMag.bVEH2Occupied:= FALSE;
		p_tyAGVToDTMag.bVEH3Occupied:= FALSE;
		p_tyAGVToDTMag.bVEHRunning	:= FALSE;

	END_IF

	bAIVInPos := p_tyAGVToDTMag.bVEHInPos1;
	bAIVAuto := p_tyAGVToDTMag.bVEHAuto;
	bAIVOccupied := p_tyAGVToDTMag.bVEH1Occupied;
	bMagConvAuto := tyDTMagToAGV.bCI1Auto;
	bMagConvOccupied :=  tyDTMagToAGV.bCI1Occupied;

	tyDTMagToAGV.bCI1Running := bMagConvRun;
	tyDTMagToAGV.bCI1Rdy	:= bMagConvRdy;

	IF p_bNtParamAGVInPosSenPrep THEN
		fbInPosErrTimer(IN:= p_tyLinkAGVtoDTMag.bVEHInPos1 AND bAGVInPosSen = FALSE, PT:= T#10s);
		IF fbInPosErrTimer.Q THEN
			eStatus		:= Error;
			udiStatus	:= 10009;	//AIV Not In Position
		END_IF
	END_IF

	IF p_bNtParamAGVInPosSenPrep THEN
		bAGVInPosSen := p_bAGVInPosSen1 AND p_bAGVInPosSen2;
	ELSE
		bAGVInPosSen := TRUE;
	END_IF

END_ACTION
```

#### Init.st
```iecst
(** 2019-01-20 **)
PROGRAM _INIT

	(* Always Change If Project Change *)

	sProgNm	:= 'AGVMag 1';

	//Physical Configuration

	//Pass Address To Global Address For External Use
	//Action, State & Status
	p_AGVMag1Stat		:= ADR(eStat);
	p_AGVMag1Status		:= ADR(eStatus);
	p_AGVMag1StatTxt	:= ADR(sStatTxt);

	//Alarm
	p_AGVMag1AlmData	:= ADR(tyAlmData);

	//Output
	p_AGVMag1RdyEnter		:= ADR(bRdyEnt);
	p_AGVMag1RdyExit		:= ADR(bRdyExit);
	p_AGVMag1McRunRdy		:= ADR(bMcRunRdy);
	p_AGVMag1DTMagToAGV		:= ADR(tyDTMagToAGV);

	(* Always Change If Project Change *)

END_PROGRAM
```

### Program Logical/AGVCom/AGV2 (IEC) - 1.00.0 - NtSMEMA v5.00.0

#### Act_InitGlobal.st
```iecst
(** 2018-12-08 **)
ACTION Act_InitGlobal:

	(* Always Change If Project Change *)

	//Pass Data To Link
	p_bLinkOpsRun ACCESS p_OpsRun;

	p_tyLinkBufferStat ACCESS p_Buffer2BffrStat;
	p_bLinkAGVOnline ACCESS p_AGVOnline;
	p_tyLinkAGVtoDTMag ACCESS p_AGVTagAGVToDTMag;

	//Pass Data To Internal Use
	p_eAct ACCESS p_OpsMagConvLD2AGVMagAct;
	p_udiRstErr	ACCESS p_RstErrReset;
	p_bPrep ACCESS p_NtParamProjAGVPrep;
	p_sProgNm ACCESS p_NtParamAGVMag2ProgNm;
	p_diTxInTimeOut ACCESS p_McParamMag2ConvRunTmOut;
	p_diTxOutTimeOut ACCESS p_McParamMag2ConvRunTmOut;
	p_eDirection ACCESS p_NtParamProjMagConvDir;
	p_bBufferMagPresent ACCESS p_DIMagPresentSen2;
	p_bMagConvLftSen ACCESS p_DIMagConvEntSen2;
	p_bMagConvRgtSen ACCESS p_DIMagPresentSen2;
	p_bMagConvMtrIn ACCESS p_MagConv2Clp2MtrSigOnOrLToR;
	p_bMagConvMtrOut ACCESS p_MagConv2Clp2MtrDirOrRToL;
	p_bNtSettingsLoadDone ACCESS p_StartupNtSettingsLoadDone;
	p_bAGVInPosSen1	ACCESS p_DIMag2AGVInPosSen1;
	p_bAGVInPosSen2	ACCESS p_DIMag2AGVInPosSen2;
	p_bNtParamAGVInPosSenPrep ACCESS p_NtParamProjAGVInPosSenPrep;
	p_bSOTRcvOk ACCESS p_DISOT2Receive;
	p_bSOTErr ACCESS p_DISOT2Error;
	p_bSOTRdy ACCESS p_DISOT2Ready;
	p_bSOTAvailable ACCESS p_DISOT2Available;
	p_bEn ACCESS p_McParamAGVComEn;
	(* Always Change If Project Change *)

END_ACTION
```

#### Act_Link.st
```iecst
(** 2018-12-08 **)
ACTION Act_Link:

	//Machine --> AGV ---> Communication On & Machine itself RUN Mode
	IF p_bLinkOpsRun = TRUE THEN

		tyDTMagToAGV.bCI2Auto := TRUE;
	ELSE
		tyDTMagToAGV.bCI2Auto	:= FALSE;
	END_IF

	tyDTMagToAGV.bCI2Occupied 			:= p_bBufferMagPresent OR p_bMagConvLftSen OR p_bMagConvRgtSen ;

	fbMagEmptyTm(IN:= p_bMagConvLftSen = FALSE AND p_bBufferMagPresent = FALSE);
	IF p_bBufferMagPresent AND p_tyLinkBufferStat.bBffrMty THEN
		tyDTMagToAGV.bCI2MagazineEmpty		:=  TRUE;
	ELSIF fbMagEmptyTm.Q THEN
		tyDTMagToAGV.bCI2MagazineEmpty		:=  FALSE;
	END_IF

	IF p_bLinkAGVOnline THEN

		p_tyAGVToDTMag.bVEHAuto		:= p_tyLinkAGVtoDTMag.bVEHAuto;
		p_tyAGVToDTMag.bVEHInPos1	:= p_tyLinkAGVtoDTMag.bVEHInPos1;
		p_tyAGVToDTMag.bVEHInPos2 	:= p_tyLinkAGVtoDTMag.bVEHInPos2 AND bAGVInPosSen;
		p_tyAGVToDTMag.bVEHInPos3 	:= p_tyLinkAGVtoDTMag.bVEHInPos3;
		p_tyAGVToDTMag.bVEH1Occupied	:= p_tyLinkAGVtoDTMag.bVEH1Occupied;
		p_tyAGVToDTMag.bVEH2Occupied	:= p_tyLinkAGVtoDTMag.bVEH2Occupied;
		p_tyAGVToDTMag.bVEH3Occupied	:= p_tyLinkAGVtoDTMag.bVEH3Occupied;
		p_tyAGVToDTMag.bVEHRunning	:= p_tyLinkAGVtoDTMag.bVEHRunning;

	ELSE

		p_tyAGVToDTMag.bVEHAuto		:= FALSE;
		p_tyAGVToDTMag.bVEHInPos1	:= FALSE;
		p_tyAGVToDTMag.bVEHInPos2 	:= FALSE;
		p_tyAGVToDTMag.bVEHInPos3 	:= FALSE;
		p_tyAGVToDTMag.bVEH1Occupied:= FALSE;
		p_tyAGVToDTMag.bVEH2Occupied:= FALSE;
		p_tyAGVToDTMag.bVEH3Occupied:= FALSE;
		p_tyAGVToDTMag.bVEHRunning	:= FALSE;

	END_IF

	bAIVInPos := p_tyAGVToDTMag.bVEHInPos2;
	bAIVAuto := p_tyAGVToDTMag.bVEHAuto;
	bAIVOccupied := p_tyAGVToDTMag.bVEH2Occupied;
	bMagConvAuto := tyDTMagToAGV.bCI2Auto;
	bMagConvOccupied :=  tyDTMagToAGV.bCI2Occupied;

	tyDTMagToAGV.bCI2Running := bMagConvRun;
	tyDTMagToAGV.bCI2Rdy	:= bMagConvRdy;

	IF p_bNtParamAGVInPosSenPrep THEN
		fbInPosErrTimer(IN:= p_tyLinkAGVtoDTMag.bVEHInPos2 AND bAGVInPosSen = FALSE, PT:= T#10s);
		IF fbInPosErrTimer.Q THEN
			eStatus		:= Error;
			udiStatus	:= 10009;	//AIV Not In Position
		END_IF
	END_IF

	IF p_bNtParamAGVInPosSenPrep THEN
		bAGVInPosSen := p_bAGVInPosSen1 AND p_bAGVInPosSen2;
	ELSE
		bAGVInPosSen := TRUE;
	END_IF

END_ACTION
```

#### Init.st
```iecst
(** 2019-01-20 **)
PROGRAM _INIT

	(* Always Change If Project Change *)

	sProgNm	:= 'AGVMag 2';

	//Physical Configuration

	//Pass Address To Global Address For External Use
	//Action, State & Status
	p_AGVMag2Stat		:= ADR(eStat);
	p_AGVMag2Status		:= ADR(eStatus);
	p_AGVMag2StatTxt	:= ADR(sStatTxt);

	//Alarm
	p_AGVMag2AlmData	:= ADR(tyAlmData);

	//Output
	p_AGVMag2RdyEnter		:= ADR(bRdyEnt);
	p_AGVMag2RdyExit		:= ADR(bRdyExit);
	p_AGVMag2McRunRdy		:= ADR(bMcRunRdy);
	p_AGVMag2DTMagToAGV		:= ADR(tyDTMagToAGV);

	(* Always Change If Project Change *)

END_PROGRAM
```

### Program Logical/AGVCom/AGV3 (IEC) - 1.00.0 - NtSMEMA v5.00.0

#### InputRef.var
```iecst
(*2019-01-20*)
(**)
(*General*)
VAR
	p_eAct : REFERENCE TO eAGVMagAction;
	p_udiRstErr : REFERENCE TO UDINT;
	p_bPrep : REFERENCE TO BOOL;
	p_bEn : REFERENCE TO BOOL;
	p_bDis : REFERENCE TO BOOL;
END_VAR
(**)
(*Configuration*)
VAR
	p_sProgNm : REFERENCE TO STRING[15];
	p_bNtSettingsLoadDone : REFERENCE TO BOOL;
	p_diTxInTimeOut : REFERENCE TO DINT;
	p_diTxOutTimeOut : REFERENCE TO DINT;
	p_eDirection : REFERENCE TO eConvDir;
END_VAR
(**)
(*Input*)
VAR
	p_tyAGVToDTMag : REFERENCE TO tyTagAGVToDTMag;
	p_bBufferMagPresent : REFERENCE TO BOOL;
	p_bNtParamAGVInPosSenPrep : REFERENCE TO BOOL;
	p_bAGVInPosSen1 : REFERENCE TO BOOL;
	p_bAGVInPosSen2 : REFERENCE TO BOOL;
	p_bMagConvLftSen : REFERENCE TO BOOL;
	p_bMagConvRgtSen : REFERENCE TO BOOL;
	p_bMagConvMtrIn : REFERENCE TO BOOL;
	p_bMagConvMtrOut : REFERENCE TO BOOL;
	p_bSOTRcvOk : REFERENCE TO BOOL;
	p_bSOTErr : REFERENCE TO BOOL;
	p_bSOTRdy : REFERENCE TO BOOL;
	p_bSOTAvailable : REFERENCE TO BOOL;
END_VAR
```

#### Local.var
```iecst
(*2019-01-20*)
(**)
(*Local Action, State & Status*)
VAR
	eAct : eAGVMagAction := AGVMagActIdle;
	eStat : eAGVMagAction := AGVMagActIdle;
	eStatus : eFBStatus := Idle;
	udiStatus : UDINT := 0;
	sStatTxt : STRING[100] := '';
	a_sStatText : ARRAY[0..50] OF STRING[100] := ['Idling','AGV Magazine Ready Enter And Communicating AGV','AGV Magazine Ready Exit And Communicating AGV',48('')];
END_VAR
(**)
(*Local Alarm*)
VAR
	tyAlmData : tyAlmDat;
	a_tyAlmText : ARRAY[10000..10099] OF tyAlmTxt := [(sAlmText:='Magazine Is Present Before Entering',sRcyText:='Remove Magazine To Continue Operation.'),(sAlmText:='AGV Not In Enter Position',sRcyText:='Adjust AGV Position And Restart Operation.'),(sAlmText:='Transfer In Time Out While Transporting',sRcyText:='Adjust Magazine Position Or Transporting Time Or Check Online Connection'),(sAlmText:='Magazine Is Not Present Before Exiting',sRcyText:='Magazine Has Taken Away, Restart Operation.'),(sAlmText:='AGV Not In Exit Position',sRcyText:='Adjust AGV Position And Restart Operation.'),(sAlmText:='Transfer Out Time Out While Transporting',sRcyText:='Adjust Magazine Position Or Transporting Time.'),(sAlmText:='AGV is not in Auto',sRcyText:='Make Sure AGV is in Auto'),(sAlmText:='Magazine is not Present in AGV while Entering',sRcyText:='Check AGV'),(sAlmText:='Magazine is Present in AGV while Exiting',sRcyText:='Check AGV'),(sAlmText:='AGV In Position Sensor is off while received the AGV in position signal',sRcyText:='Check AGV in position sensor'),(sAlmText:='SOT Error Signal Has Been Activated',sRcyText:='AIV Activated The Error Signal During Magazine Transportation'),89((0))];
END_VAR
(**)
(*Local Output*)
VAR
	bMcRunRdy : BOOL;
	bRdyEnt : BOOL;
	bRdyExit : BOOL;
	bMagEnt : BOOL;
	bMagExit : BOOL;
END_VAR
(**)
(*Local Input*)
VAR
	udiRstErr : UDINT := 0;
	bPrep : BOOL := TRUE;
	bEn : BOOL := TRUE;
	bDis : BOOL := FALSE;
	sProgNm : STRING[15] := 'AGVMag';
	bNtSettingsLoadDone : BOOL := TRUE;
	diTxInTimeOut : DINT;
	diTxOutTimeOut : DINT;
	eDirection : eConvDir;
	bBufferMagPresent : BOOL;
	bMagConvLftSen : BOOL;
	bMagConvRgtSen : BOOL;
	bMagConvMtrIn : BOOL;
	bMagConvMtrOut : BOOL;
	bAGVInSen1 : BOOL;
	bAGVInSen2 : BOOL;
	bNtParamAGVInPosSenPrep : BOOL;
	tyAGVToDTMag : tyTagAGVToDTMag;
	tyDTMagToAGV : tyTagDTMagToAGV;
END_VAR
(**)
(*Local*)
VAR
	bRstErr : BOOL;
	udiRstErrOld : UDINT;
	bInitDone : BOOL;
	bInitialDone : BOOL;
	usiStep : USINT;
	bEndSen : BOOL;
	bAGVInPosSen : BOOL;
	fbMagEmptyTm : TON := (PT:=T#2s);
	fbInPosErrTimer : TON;
	fbTxInTimer : TON;
	fbTxOutTimer : TON;
	fbMagOutTrig : F_TRIG;
	eStatOld : eAGVMagAction := AGVMagActIdle;
	fbCheckErrorTim : TON := (PT:=T#1s);
	bMagConvRun : BOOL;
	bMagConvRdy : BOOL;
	bMagConvAuto : BOOL;
	bMagConvOccupied : BOOL;
	bAIVOccupied : BOOL;
	bAIVAuto : BOOL;
	bAIVInPos : BOOL;
	udiModuleNum : UDINT := 6161;
END_VAR
```

#### Act_InitGlobal.st
```iecst
(** 2018-12-08 **)
ACTION Act_InitGlobal:

	(* Always Change If Project Change *)

	//Pass Data To Link
	p_bLinkOpsRun ACCESS p_OpsRun;
	p_tyLinkBufferStat ACCESS p_Buffer3BffrStat;
	p_bLinkAGVOnline ACCESS p_AGVOnline;
	p_tyLinkAGVtoDTMag ACCESS p_AGVTagAGVToDTMag;

	//Pass Data To Internal Use
	p_eAct ACCESS p_OpsMagConvLD3AGVMagAct;
	p_udiRstErr	ACCESS p_RstErrReset;
	p_bPrep ACCESS p_NtParamProjAGVPrep;
	p_sProgNm ACCESS p_NtParamAGVMag3ProgNm;
	p_diTxInTimeOut ACCESS p_McParamMag3ConvRunTmOut;
	p_diTxOutTimeOut ACCESS p_McParamMag3ConvRunTmOut;
	p_eDirection ACCESS p_NtParamProjMagConvDir;
	p_bBufferMagPresent ACCESS p_DIMagPresentSen3;
	p_bMagConvLftSen ACCESS p_DIMagConvEntSen3;
	p_bMagConvRgtSen ACCESS p_DIMagPresentSen3;
	p_bMagConvMtrIn ACCESS p_MagConv2Clp3MtrSigOnOrLToR;
	p_bMagConvMtrOut ACCESS p_MagConv2Clp3MtrDirOrRToL;
	p_bNtSettingsLoadDone ACCESS p_StartupNtSettingsLoadDone;
	p_bAGVInPosSen1	ACCESS p_DIMag3AGVInPosSen1;
	p_bAGVInPosSen2	ACCESS p_DIMag3AGVInPosSen2;
	p_bNtParamAGVInPosSenPrep ACCESS p_NtParamProjAGVInPosSenPrep;
	p_bSOTRcvOk ACCESS p_DISOT3Receive;
	p_bSOTErr ACCESS p_DISOT3Error;
	p_bSOTRdy ACCESS p_DISOT3Ready;
	p_bSOTAvailable ACCESS p_DISOT3Available;
	p_bEn ACCESS p_McParamAGVComEn;
	(* Always Change If Project Change *)

END_ACTION
```

#### Act_InitLocal.st
```iecst
(** 2019-01-20 **)
ACTION Act_InitLocal:

	//Input Reference Link To Local Variable
	p_eAct ACCESS ADR(eAct);
	p_udiRstErr ACCESS ADR(udiRstErr);
	p_bPrep ACCESS ADR(bPrep);
	p_bEn ACCESS ADR(bEn);
	p_bDis ACCESS ADR(bDis);
	p_sProgNm ACCESS ADR(sProgNm);
	p_tyAGVToDTMag ACCESS ADR(tyAGVToDTMag);
	p_bNtSettingsLoadDone ACCESS ADR(bNtSettingsLoadDone);
	p_diTxInTimeOut ACCESS ADR(diTxInTimeOut);
	p_diTxOutTimeOut ACCESS ADR(diTxOutTimeOut);
	p_eDirection ACCESS ADR(eDirection);
	p_bBufferMagPresent ACCESS ADR(bBufferMagPresent);
	p_bMagConvLftSen ACCESS ADR(bMagConvLftSen);
	p_bMagConvRgtSen ACCESS ADR(bMagConvRgtSen);
	p_bMagConvMtrIn ACCESS ADR(bMagConvMtrIn);
	p_bMagConvMtrOut ACCESS ADR(bMagConvMtrOut);
	p_bAGVInPosSen1 ACCESS ADR(bAGVInSen1);
	p_bAGVInPosSen2 ACCESS ADR(bAGVInSen2);
	p_bNtParamAGVInPosSenPrep ACCESS ADR(bNtParamAGVInPosSenPrep);
END_ACTION
```

#### Act_Link.st
```iecst
(** 2018-12-08 **)
ACTION Act_Link:

	//Machine --> AGV ---> Communication On & Machine itself RUN Mode
	IF p_bLinkOpsRun = TRUE THEN

		tyDTMagToAGV.bCI3Auto := TRUE;
	ELSE
		tyDTMagToAGV.bCI3Auto	:= FALSE;
	END_IF

	tyDTMagToAGV.bCI3Occupied 			:= p_bBufferMagPresent OR p_bMagConvLftSen OR p_bMagConvRgtSen ;

	fbMagEmptyTm(IN:= p_bMagConvLftSen = FALSE AND p_bBufferMagPresent = FALSE);
	IF p_bBufferMagPresent AND p_tyLinkBufferStat.bBffrMty THEN
		tyDTMagToAGV.bCI3MagazineEmpty		:=  TRUE;
	ELSIF fbMagEmptyTm.Q THEN
		tyDTMagToAGV.bCI3MagazineEmpty		:=  FALSE;
	END_IF

	IF p_bLinkAGVOnline THEN

		p_tyAGVToDTMag.bVEHAuto		:= p_tyLinkAGVtoDTMag.bVEHAuto;
		p_tyAGVToDTMag.bVEHInPos1	:= p_tyLinkAGVtoDTMag.bVEHInPos1;
		p_tyAGVToDTMag.bVEHInPos2 	:= p_tyLinkAGVtoDTMag.bVEHInPos2;
		p_tyAGVToDTMag.bVEHInPos3 	:= p_tyLinkAGVtoDTMag.bVEHInPos3 AND bAGVInPosSen;
		p_tyAGVToDTMag.bVEH1Occupied	:= p_tyLinkAGVtoDTMag.bVEH1Occupied;
		p_tyAGVToDTMag.bVEH2Occupied	:= p_tyLinkAGVtoDTMag.bVEH2Occupied;
		p_tyAGVToDTMag.bVEH3Occupied	:= p_tyLinkAGVtoDTMag.bVEH3Occupied;
		p_tyAGVToDTMag.bVEHRunning	:= p_tyLinkAGVtoDTMag.bVEHRunning;

	ELSE

		p_tyAGVToDTMag.bVEHAuto		:= FALSE;
		p_tyAGVToDTMag.bVEHInPos1	:= FALSE;
		p_tyAGVToDTMag.bVEHInPos2 	:= FALSE;
		p_tyAGVToDTMag.bVEHInPos3 	:= FALSE;
		p_tyAGVToDTMag.bVEH1Occupied:= FALSE;
		p_tyAGVToDTMag.bVEH2Occupied:= FALSE;
		p_tyAGVToDTMag.bVEH3Occupied:= FALSE;
		p_tyAGVToDTMag.bVEHRunning	:= FALSE;

	END_IF

	bAIVInPos := p_tyAGVToDTMag.bVEHInPos3;
	bAIVAuto := p_tyAGVToDTMag.bVEHAuto;
	bAIVOccupied := p_tyAGVToDTMag.bVEH3Occupied;
	bMagConvAuto := tyDTMagToAGV.bCI3Auto;
	bMagConvOccupied :=  tyDTMagToAGV.bCI3Occupied;

	tyDTMagToAGV.bCI3Running := bMagConvRun;
	tyDTMagToAGV.bCI3Rdy	:= bMagConvRdy;

	IF p_bNtParamAGVInPosSenPrep THEN
		fbInPosErrTimer(IN:= p_tyLinkAGVtoDTMag.bVEHInPos3 AND bAGVInPosSen = FALSE, PT:= T#10s);
		IF fbInPosErrTimer.Q THEN
			eStatus		:= Error;
			udiStatus	:= 10009;	//AIV Not In Position
		END_IF
	END_IF

	IF p_bNtParamAGVInPosSenPrep THEN
		bAGVInPosSen := p_bAGVInPosSen1 AND p_bAGVInPosSen2;
	ELSE
		bAGVInPosSen := TRUE;
	END_IF

END_ACTION
```

#### Act_LinkAction.st
```iecst
(** 2019-03-29 **)
ACTION Act_LinkAction:

	IF EDGENEG (p_bLinkOpsRun) THEN
		p_eAct	:= AGVMagActIdle;
	END_IF

END_ACTION
```

### AGV4.var - Change By Project
```iecst
(*2019-01-20*)
(**)
(*Action & State & Status*)
VAR
	p_AGVMag4Stat : UDINT;
	p_AGVMag4Status : UDINT;
	p_AGVMag4StatTxt : UDINT;
END_VAR
(**)
(*Alarm*)
VAR
	p_AGVMag4AlmData : UDINT;
END_VAR
(**)
(*Output*)
VAR
	p_AGVMag4RdyEnter : UDINT;
	p_AGVMag4RdyExit : UDINT;
	p_AGVMag4McRunRdy : UDINT;
	p_AGVMag4Exit : UDINT;
	p_AGVMag4DTMagToAGV : UDINT;
END_VAR
```

### Program Logical/AGVCom/AGV4 (IEC) - 1.00.0 - NtSMEMA v5.00.0

#### InputRef_Link.var
```iecst
(*2018-12-08*)
(**)
(*External Data*)
VAR
	p_bLinkOpsRun : REFERENCE TO BOOL;
END_VAR
(**)
VAR
	p_tyLinkBufferStat : REFERENCE TO tyBffrStat;
	p_bLinkAGVOnline : REFERENCE TO BOOL;
	p_tyLinkAGVtoDTMag : REFERENCE TO tyTagAGVToDTMag;
END_VAR
```

#### Act_Alarm.st
```iecst
(** 2019-03-25 **)
ACTION Act_Alarm:

	//Error
	IF EDGEPOS(eStatus = Error) THEN

		tyAlmData.sProgNm		:= p_sProgNm;
		tyAlmData.udiCode		:= udiStatus;
		tyAlmData.eSeverity		:= AlmSeverityError;
		tyAlmData.udiRunTime	:= tyAlmData.udiRunTime + 1;
		tyAlmData.bAlm			:= TRUE;
		tyAlmData.udiModuleNum  := udiModuleNum;
		g_sAGVProgNm		:= p_sProgNm;
		//Get Error Message
		IF tyAlmData.udiCode < 10000 OR tyAlmData.udiCode > 10099 THEN
			tyAlmData.sAlmMsg	:= 'Unknown';
			tyAlmData.sRcyMsg	:= 'Unknown';
		ELSE
			tyAlmData.sAlmMsg	:= a_tyAlmText[tyAlmData.udiCode].sAlmText;
			tyAlmData.sRcyMsg	:= a_tyAlmText[tyAlmData.udiCode].sRcyText;
		END_IF

		sStatTxt	:= tyAlmData.sAlmMsg;

	ELSIF bRstErr AND (tyAlmData.udiCode <> 0) THEN

		tyAlmData.udiCode	:= 0;
		tyAlmData.eSeverity	:= AlmSeverityNA;
		tyAlmData.sAlmMsg	:= '';
		tyAlmData.sRcyMsg	:= '';
		tyAlmData.bAlm			:= FALSE;
		sStatTxt	:= a_sStatText[eStat];

	END_IF

END_ACTION
```

#### Act_InitGlobal.st
```iecst
(** 2021-05-31 **)
ACTION Act_InitGlobal:

	(* Always Change If Project Change *)

	//Pass Data To Link
	p_bLinkOpsRun ACCESS p_OpsRun;
	p_tyLinkBufferStat ACCESS p_Buffer4BffrStat;
	p_bLinkAGVOnline ACCESS p_AGVOnline;
	p_tyLinkAGVtoDTMag ACCESS p_AGVTagAGVToDTMag;

	//Pass Data To Internal Use
	p_eAct ACCESS p_OpsMagConvLD4AGVMagAct;
	p_udiRstErr	ACCESS p_RstErrReset;
	p_bPrep ACCESS p_NtParamProjAGVPrep;
	p_sProgNm ACCESS p_NtParamAGVMag4ProgNm;
	p_diTxInTimeOut ACCESS p_McParamMag4ConvRunTmOut;
	p_diTxOutTimeOut ACCESS p_McParamMag4ConvRunTmOut;
	p_eDirection ACCESS p_NtParamProjMagConvDir;
	p_bBufferMagPresent ACCESS p_DIMagPresentSen4;
	p_bMagConvLftSen ACCESS p_DIMagConvEntSen4;
	p_bMagConvRgtSen ACCESS p_DIMagPresentSen4;
	p_bMagConvMtrIn ACCESS p_MagConv2Clp4MtrSigOnOrLToR;
	p_bMagConvMtrOut ACCESS p_MagConv2Clp4MtrDirOrRToL;
	p_bNtSettingsLoadDone ACCESS p_StartupNtSettingsLoadDone;
	p_bAGVInPosSen1	ACCESS p_DIMag4AGVInPosSen1;
	p_bAGVInPosSen2	ACCESS p_DIMag4AGVInPosSen2;
	p_bNtParamAGVInPosSenPrep ACCESS p_NtParamProjAGVInPosSenPrep;
	p_bSOTRcvOk ACCESS p_DISOT4Receive;
	p_bSOTErr ACCESS p_DISOT4Error;
	p_bSOTRdy ACCESS p_DISOT4Ready;
	p_bSOTAvailable ACCESS p_DISOT4Available;
	p_bEn ACCESS p_McParamAGVComEn;
	(* Always Change If Project Change *)

END_ACTION
```
